					// Filebuffer Offset increment
					pstSysInfo^.stFileHandler.udiTmpFileBufferOffset := pstSysInfo^.stFileHandler.udiTmpFileBufferOffset + pstSysInfo^.udiTmpRecordLen;
					
					// clear temp. record buffer
					pstSysInfo^.bolTmpRecordFull := FALSE;
					
					// Record Buffer ist frei -> Offset zu Null setzen
					pstSysInfo^.udiTmpRecordLen := 0;
				END_IF
			ELSE // file buffer + temp record buffer exceeds maximum
				pstSysInfo^.stFileHandler.udiWriteTimer := 0; // reset timer
				pstSysInfo^.stFileHandler.usiCmd := FileLc.cCMD_FLUSHBUF; // write file buffer to file
			END_IF
		END_IF
		
		// return if buffer still full
		IF (pstSysInfo^.bolTmpRecordFull) THEN
			RETURN;
		END_IF
			

		// reset flag
		bolWriteRecord := FALSE;
		
		// Read out from base log -> stData
		uinReadStatus := stFileLogClientLibInfo.p_fbBasLog^.M_Read(In_pHandle:=pstSysInfo^.pBaseLogHandle,In_pData:=ADR(stData)); 
		IF (uinReadStatus<>0) THEN // exit for if nothing to read
			RETURN;
		END_IF
	
		// base logging
		IF(pstSysInfo^.uinLogTyp=FileLc.cLOGTYP_BL) THEN
			//reference item list
			pstItemCfgList := pstSysInfo^.stItemInfo.p_bytItemCfgList;
			
			// on BL only use first line
			pstItemDataList := pstSysInfo^.stItemInfo.a_p_bytItemDataList[0];
			
			// must be worked on the PvId ?
			 FOR jj := 0 TO (pstSysInfo^.stItemInfo.uinActNbrOfItems-1) BY 1 DO
				 CASE (pstItemCfgList[jj].dinPvId) OF
					FileLc.cPVTYPE_BL_LOGTYP:
						M_WriteActItemIdx(In_pstItemDataList :=pstItemDataList,In_dinDataTyp:= FileLc.cVAR_TYPE_UDINT, In_pValue:=ADR(stData.udiLogType), In_udiRecIdx:=0, In_uinActItemIdx:=jj);
					FileLc.cPVTYPE_BL_CTRL_ID:
						M_WriteActItemIdx(In_pstItemDataList :=pstItemDataList,In_dinDataTyp:= FileLc.cVAR_TYPE_INT, In_pValue:=ADR(stData.intCtrlID), In_udiRecIdx:=0, In_uinActItemIdx:=jj);
					FileLc.cPVTYPE_BL_STRING1:
						M_WriteActItemIdx(In_pstItemDataList :=pstItemDataList,In_dinDataTyp:= FileLc.cVAR_TYPE_STRING, In_pValue:=ADR(stData.strText1), In_udiRecIdx:=0, In_uinActItemIdx:=jj);
					FileLc.cPVTYPE_BL_STRING2:
						M_WriteActItemIdx(In_pstItemDataList :=pstItemDataList,In_dinDataTyp:= FileLc.cVAR_TYPE_STRING, In_pValue:=ADR(stData.strText2), In_udiRecIdx:=0, In_uinActItemIdx:=jj);
					FileLc.cPVTYPE_BL_PAR1:
						M_WriteActItemIdx(In_pstItemDataList :=pstItemDataList,In_dinDataTyp:= FileLc.cVAR_TYPE_DINT, In_pValue:=ADR(stData.dinPar1), In_udiRecIdx:=0, In_uinActItemIdx:=jj);
					FileLc.cPVTYPE_BL_PAR2:
						M_WriteActItemIdx(In_pstItemDataList :=pstItemDataList,In_dinDataTyp:= FileLc.cVAR_TYPE_DINT, In_pValue:=ADR(stData.dinPar2), In_udiRecIdx:=0, In_uinActItemIdx:=jj);
					FileLc.cPVTYPE_BL_PAR3:
						M_WriteActItemIdx(In_pstItemDataList :=pstItemDataList,In_dinDataTyp:= FileLc.cVAR_TYPE_DINT, In_pValue:=ADR(stData.dinPar3), In_udiRecIdx:=0, In_uinActItemIdx:=jj);
					FileLc.cPVTYPE_BL_PAR4:
						M_WriteActItemIdx(In_pstItemDataList :=pstItemDataList,In_dinDataTyp:= FileLc.cVAR_TYPE_DINT, In_pValue:=ADR(stData.dinPar4), In_udiRecIdx:=0, In_uinActItemIdx:=jj);
							
				END_CASE
			 END_FOR
			 // general inf o add to Record list
			pstSysInfo^.stItemInfo.stItemRecordData[0].dtActDateTime := stData.dtDateTimeEntry;
			pstSysInfo^.stItemInfo.stItemRecordData[0].uinActMilli := stData.uinMs;
			
			// for BaseLog write always record 0
			M_WriteRecord(In_pstSysInfo:=pstSysInfo,In_uinItemListIdx := 0);
			
			// end of IF(pstSysInfo^.uinLogTyp=FileLc.cLOGTYP_BL) THEN
		ELSE
			(* -----------------------------------*/
		  /* Data- und PV - Logging             */
		  /* -----------------------------------*)
	
		  (* ----------------------*/
		  /* Check commandes     */
		  /* ----------------------
		  /* "cmd" in typ field *)
		  IF (stData.dinPar3 = BasLog.cVAR_TYPE_CMD_NEW_REC) THEN
	
				(* search free record - list *)
				FOR jj := 0 TO Queue.cMAX_NR_OF_TASKS BY 1 DO
				  IF ((pstSysInfo^.stItemInfo.stItemRecordData[jj].udiRecIdx = 0) OR (DINT_TO_UDINT(stData.dinPar4) = pstSysInfo^.stItemInfo.stItemRecordData[jj].udiRecIdx)) THEN
						pstSysInfo^.stItemInfo.stItemRecordData[jj].udiRecIdx := DINT_TO_UDINT(stData.dinPar4);
						pstSysInfo^.stItemInfo.stItemRecordData[jj].dtActDateTime := stData.dtDateTimeEntry;
						pstSysInfo^.stItemInfo.stItemRecordData[jj].uinActMilli := stData.uinMs;
						EXIT;
				  END_IF
			   END_FOR
		  
		  ELSIF (stData.dinPar3 = BasLog.cVAR_TYPE_CMD_END_REC) THEN
			bolWriteRecord := TRUE;
		  END_IF			
	
	
		  (* --------------------------------------------------------------*/
		  /* entry reached BaseLog message in record list */
		  /* --------------------------------------------------------------*)
		  M_PutPvIdInList(In_pstSysInfo := pstSysInfo, In_pstData := ADR(stData));
	
		  (* -----------------------------------------------------*/
		  /* write the complete record to the temporar buffer */
		  /* -----------------------------------------------------*)
		  IF (bolWriteRecord)  THEN
			FOR jj := 0 TO Queue.cMAX_NR_OF_TASKS BY 1 DO
			  (* Is the reached record index allready entried in referencelist *)
			  IF (pstSysInfo^.stItemInfo.stItemRecordData[jj].udiRecIdx = DINT_TO_UDINT(stData.dinPar4)) THEN
				M_WriteRecord(In_pstSysInfo:=pstSysInfo,In_uinItemListIdx := jj);
				EXIT;
			  END_IF
			END_FOR
		  END_IF
    END_IF // else
  END_FOR // FOR ii := 0 TO ((pstSysInfo^.stItemInfo.uinActNbrOfItems-1) * 20) BY 1 DO
END_IF 	//IF (pstSysInfo^.stItemInfo.uinActNbrOfItems>0) THEN
END_METHOD

METHOD PUBLIC M_Init : BOOL
VAR_INPUT
	In_strCfgFileName: STRING(FileLc.cFILENAME_LENGTH); // name of the config/template file
	In_strPath: STRING(FileLc.cPATH_LENGTH);  // path of the config/template file
	In_p_fbBasLog: POINTER TO FB_BasLog; // only one central FB_BasLog instance allowed per PLC!!!
	In_bolExecute : BOOL;
	In_p_uinFLcIdx : POINTER TO UINT; // actual file client id
END_VAR
VAR_OUTPUT
	Out_pHandle: POINTER TO T_FileLc_SysInfo; // handle for cyclic call	
	Out_udiStatus: UDINT; 	// 0 => successful done, <>0 => error
	Out_bolDone: BOOL;		// Done
END_VAR

VAR
	strClientName : STRING(255);
	uinFLcIdxForArr : UINT;
	udiStatus : UDINT;
	udiMask : UDINT;
	uinInitStatus : UINT;
	pQueueInfoHandle : POINTER TO POINTER TO T_Queue_Info;
	fbGETCURTASKINDEX: Tc2_System.GETCURTASKINDEX;
	udiTaskCnt : UDINT;
END_VAR
// only one client init at the same on PLC possibel!!!
IF (In_p_uinFLcIdx<>Tc3_MemMan.NULL) THEN // valid actual id reference
	IF (In_bolExecute=TRUE) THEN
		// wait until release init rom other clients...
		IF  ((stFileLogClientLibInfo.uinActClientInitActive=0) OR (stFileLogClientLibInfo.uinActClientInitActive=In_p_uinFLcIdx^)) THEN
			IF (stFileLogClientLibInfo.uinActClientInitActive=0) THEN
				stFileLogClientLibInfo.uinActClientInitActive := stFileLogClientLibInfo.uinActNbrOfFileClients + 1; // lock init of other clients!!!
				In_p_uinFLcIdx^ := stFileLogClientLibInfo.uinActClientInitActive;
				
				Out_bolDone := 0;
				Out_udiStatus := 0;
				Out_pHandle := 0;
				//reset statemachine
				(* check input parameter *)
				IF (stFileLogClientLibInfo.uinActNbrOfFileClients >= FileLc.cMAX_NBR_OF_FILECLIENTS) THEN
					Out_udiStatus := FileLc.cERR_NBR_OF_FC_EXEEDED;
					RETURN;
				END_IF
				
				IF (In_strCfgFileName='') THEN
					Out_udiStatus := FileLc.cERR_FILENAME_MISSING;
					RETURN;
				END_IF
				
				IF (In_strPath='') THEN
					Out_udiStatus := FileLc.cERR_PATH_MISSING;
					RETURN;
				END_IF
				
				IF (In_p_fbBasLog=TC3_MEMMAN.NULL) THEN
					Out_udiStatus := FileLc.cERR_NO_BASELOG;
					RETURN;
				END_IF
		
				stFileLogClientLibInfo.p_fbBasLog := In_p_fbBasLog;
				
				// actual client init
				stFileLogClientLibInfo.stSysInfo[stFileLogClientLibInfo.uinActNbrOfFileClients].stStatemachine.uinState := 1;
				stFileLogClientLibInfo.stSysInfo[stFileLogClientLibInfo.uinActNbrOfFileClients].stStatemachine.uinState_old := 0;
				stFileLogClientLibInfo.stSysInfo[stFileLogClientLibInfo.uinActNbrOfFileClients].fbFileLc_WorkOnFile(In_bolExecute:=FALSE); // reset statemachine on next positive edge!
				
				// increment client number
				stFileLogClientLibInfo.uinActNbrOfFileClients := stFileLogClientLibInfo.uinActNbrOfFileClients + 1;
				
				
			END_IF
		
			// valid client idx
			IF (In_p_uinFLcIdx^>0) THEN
				uinFLcIdxForArr := In_p_uinFLcIdx^-1; // access idx for arrays!
			
				CASE stFileLogClientLibInfo.stSysInfo[uinFLcIdxForArr].stStatemachine.uinState OF
					1:
						// check template/config file */
						stFileLogClientLibInfo.stSysInfo[uinFLcIdxForArr].fbFileLc_WorkOnFile(In_bolExecute:=TRUE,In_strPath:=In_strPath,In_strCfgFileName:=In_strCfgFileName,In_pstSysInfo := ADR(stFileLogClientLibInfo.stSysInfo[uinFLcIdxForArr]));
						IF (stFileLogClientLibInfo.stSysInfo[uinFLcIdxForArr].fbFileLc_WorkOnFile.Out_udiStatus<>0) OR (stFileLogClientLibInfo.stSysInfo[uinFLcIdxForArr].fbFileLc_WorkOnFile.Out_bolDone=1) THEN
							stFileLogClientLibInfo.stSysInfo[uinFLcIdxForArr].stStatemachine.uinState := 2;
						END_IF
						
					2:
						IF (stFileLogClientLibInfo.stSysInfo[uinFLcIdxForArr].fbFileLc_WorkOnFile.Out_udiStatus<>0) THEN // error in template/config file
							stFileLogClientLibInfo.uinActNbrOfFileClients := stFileLogClientLibInfo.uinActNbrOfFileClients - 1;
							Out_udiStatus := stFileLogClientLibInfo.stSysInfo[uinFLcIdxForArr].fbFileLc_WorkOnFile.Out_udiStatus;
							RETURN;
						END_IF
						  
						// register as client on base log system
						strClientName := BasLog.cCLIENT_NAME_PF;
						strClientName := Tc2_Standard.CONCAT(strClientName,'.fileclient');
						strClientName := Tc2_Standard.CONCAT(strClientName,UINT_TO_STRING(uinFLcIdxForArr));
						
						//LOG TYPE Maske --> PVLog Event und Cyclic 
						CASE (stFileLogClientLibInfo.stSysInfo[uinFLcIdxForArr].uinLogTyp) OF
							FileLc.cLOGTYP_DATA:
								udiMask := BasLog.cLOGTYPE_DATA;
							FileLc.cLOGTYP_PV:
								udiMask := (BasLog.cLOGTYPE_PV_EVENT OR BasLog.cLOGTYPE_PV_CYCLIC);
							FileLc.cLOGTYP_BL, FileLc.cLOGTYP_OPEN:
								udiMask := stFileLogClientLibInfo.stSysInfo[uinFLcIdxForArr].udiMask;
						END_CASE
						
						stFileLogClientLibInfo.fbTimeStamp.In_strNetId := stFileLogClientLibInfo.stSysInfo[uinFLcIdxForArr].stConfig.strLogNetId; // use system time of log target system
						stFileLogClientLibInfo.fbTimeStamp.In_t_CycleTimeRefreshTimeZone := T#0S; // cyclic check time zone settings - not needed using LocalTime_FileTime_BaseWin for log system and local time
						stFileLogClientLibInfo.p_fbBasLog^.M_ClientInit(In_strClientName:=strClientName,In_udiMask := udiMask, In_uinNrOfElement:= UDINT_TO_UINT(stFileLogClientLibInfo.stSysInfo[uinFLcIdxForArr].stConfig.udiQueueLen),In_p_fbTimeStamp:=ADR(stFileLogClientLibInfo.fbTimeStamp),In_bolUseLocalTimeStamp:=stFileLogClientLibInfo.stSysInfo[uinFLcIdxForArr].stConfig.bolUseLocalTimeStamp,Out_pHandle=>pQueueInfoHandle,Out_uinStatus=>udiStatus);
						
						IF (udiStatus<>0) THEN // check if init base log ok
							stFileLogClientLibInfo.uinActNbrOfFileClients := stFileLogClientLibInfo.uinActNbrOfFileClients - 1;
							Out_udiStatus := udiStatus;
							RETURN;
						END_IF
				
						//---------------------------------------------------------------------------------------------------------------
						// set SysInfo parameter
						stFileLogClientLibInfo.stSysInfo[uinFLcIdxForArr].pBaseLogHandle := pQueueInfoHandle;
						//DeviceName auf SysInfo Struktur ablegen
						stFileLogClientLibInfo.stSysInfo[uinFLcIdxForArr].strPathName := In_strPath;
						
						// get cycle time
						// number of tasksudiTaskCnt := TwinCAT_SystemInfoVarList._AppInfo.TaskCnt;
						fbGETCURTASKINDEX();
						udiTaskCnt := fbGETCURTASKINDEX.index;
						stFileLogClientLibInfo.stSysInfo[uinFLcIdxForArr].udiCylceTimeMs := TwinCAT_SystemInfoVarList._TaskInfo[UDINT_TO_DINT(udiTaskCnt)].CycleTime/10000; //[ms] X[100ns]/10000 -> [ms]
			
						// init filehandler
						//automatic read out infos about FUB
						udiStatus := stFileLogClientLibInfo.stSysInfo[uinFLcIdxForArr].stFileHandler.FB_FileLc_FileHdl.M_Init(In_pstSysInfo:=ADR(stFileLogClientLibInfo.stSysInfo[uinFLcIdxForArr]));
						IF (udiStatus<>0) THEN // check if init base log ok
							stFileLogClientLibInfo.uinActNbrOfFileClients := stFileLogClientLibInfo.uinActNbrOfFileClients - 1;
							Out_udiStatus := udiStatus;
							RETURN;
						END_IF
						
						// finished
						stFileLogClientLibInfo.stSysInfo[uinFLcIdxForArr].stStatemachine.uinState := 3;
					3:
						// wait for time stamp init ok (synchronize windows time, get time zone information!)
						stFileLogClientLibInfo.fbTimeStamp();
						IF (stFileLogClientLibInfo.fbTimeStamp.Out_bolInitOk) THEN
							stFileLogClientLibInfo.stSysInfo[uinFLcIdxForArr].stStatemachine.uinState := 4;
						END_IF
					4: 
						stFileLogClientLibInfo.stSysInfo[uinFLcIdxForArr].stStatemachine.usiInitDone := 1;
						Out_bolDone := TRUE; // init done
						stFileLogClientLibInfo.uinActClientInitActive := 0; // release init of other clients!!!
						// return adresse on actual SysInfo struct
						Out_pHandle := ADR(stFileLogClientLibInfo.stSysInfo[uinFLcIdxForArr]);
				END_CASE
			END_IF
		END_IF
	ELSE
		IF (stFileLogClientLibInfo.uinActClientInitActive=In_p_uinFLcIdx^) THEN // reset own flag
			stFileLogClientLibInfo.uinActClientInitActive := 0; // release init of other clients!!!
		END_IF
	END_IF
ELSE
	Out_pHandle := 0;
	Out_udiStatus := FileLc.cERR_NO_FLCIDX;
	RETURN;
END_IF
END_METHOD

METHOD PROTECTED M_PutPvIdInList : UINT
VAR_INPUT
	In_pstSysInfo: POINTER TO T_FileLc_SysInfo;
	In_pstData : POINTER TO T_Bl_BaseStruc;
END_VAR
VAR
	pstItemDataList : POINTER TO T_FileLc_ItemData;
  	pstItemCfgList: POINTER TO T_FileLc_ItemCfg;
	pstItemCfgListItem: T_FileLc_ItemCfg;
	bolItemFound : BOOL;
	uinActItemIdx : UINT;
	ii: UINT;
END_VAR
// Methode check received base log message and fill up the data to the item list
pstItemCfgList := In_pstSysInfo^.stItemInfo.p_bytItemCfgList;

bolItemFound := FALSE;

// has the id to be overworked?
FOR ii := 0 TO (In_pstSysInfo^.stItemInfo.uinActNbrOfItems-1) BY 1 DO
	pstItemCfgListItem := pstItemCfgList[ii];
	IF (pstItemCfgList[ii].dinPvId=In_pstData^.dinPar1) THEN
	 	bolItemFound := TRUE;
		uinActItemIdx := ii;
		EXIT;
	END_IF
END_FOR

// this PvId is not in list
IF (bolItemFound=FALSE) THEN
	M_PutPvIdInList := 0;
	RETURN;
END_IF

(* ---------------------------------*/
/* check reference list      */
/* and write data to the list */
/* ---------------------------------*)
FOR ii := 0 TO Queue.cMAX_NR_OF_TASKS BY 1 DO

	(* Is the received record in reference list?*)
	IF (In_pstSysInfo^.stItemInfo.stItemRecordData[ii].udiRecIdx = DINT_TO_UDINT(In_pstData^.dinPar4)) THEN
			
	  // reference to item list
	  pstItemDataList := In_pstSysInfo^.stItemInfo.a_p_bytItemDataList[ii];
	
	  (* write data to item list *)
	  IF (In_pstData^.dinPar3 = FileLc.cVAR_TYPE_STRING) THEN// data definition
		M_WriteActItemIdx(In_pstItemDataList :=pstItemDataList,In_dinDataTyp:= FileLc.cVAR_TYPE_STRING, In_pValue:=ADR(In_pstData^.strText2), In_udiRecIdx:=DINT_TO_UDINT(In_pstData^.dinPar4), In_uinActItemIdx:=uinActItemIdx);
	  ELSE
		M_WriteActItemIdx(In_pstItemDataList:=pstItemDataList, In_dinDataTyp := In_pstData^.dinPar3, In_pValue := ADR(In_pstData^.dinPar2),In_udiRecIdx := DINT_TO_UDINT(In_pstData^.dinPar4), In_uinActItemIdx := uinActItemIdx);
	  END_IF
	  EXIT;
	END_IF
END_FOR		

M_PutPvIdInList := 0;
RETURN;
END_METHOD

METHOD PROTECTED M_ReleaseBuffer : UINT

VAR_INPUT
	In_pReleaseBuffer : POINTER TO BYTE;
END_VAR
//delocate  allocated buffer with __NEW
__DELETE(In_pReleaseBuffer);
RETURN; // delete buffer with dynamic size...
END_METHOD

METHOD PROTECTED M_WriteActItemIdx : UINT
VAR_INPUT
	In_pstItemDataList : POINTER TO T_FileLc_ItemData;
	In_dinDataTyp: DINT;
	In_pValue: POINTER TO BYTE;
	In_udiRecIdx : UDINT;
	In_uinActItemIdx : UINT;
END_VAR

VAR
	strTmp : T_MaxString;
	pString : POINTER TO STRING(255);
	pBool : POINTER TO BOOL;
	pSint : POINTER TO SINT;
	pInt : POINTER TO INT;
	pDint : POINTER TO DINT;
	pUsint : POINTER TO USINT;
	pUint : POINTER TO UINT;
	pUdint : POINTER TO UDINT;
	pReal : POINTER TO REAL;
	pLreal : POINTER TO LREAL;
	stItemDataListItem : T_FileLc_ItemData;
END_VAR
// write value in ItemList based on datatyp
IF (In_pValue<>TC3_MEMMAN.NULL) THEN
	 CASE In_dinDataTyp OF
		FileLc.cVAR_TYPE_SINT:
			pSint := In_pValue;
			strTmp := SINT_TO_STRING(pSint^);	
		FileLc.cVAR_TYPE_INT:
			pInt := In_pValue;
			strTmp := INT_TO_STRING(pInt^);
		FileLc.cVAR_TYPE_DINT:
			pDint := In_pValue;
			strTmp := DINT_TO_STRING(pDint^);
		FileLc.cVAR_TYPE_BOOL:
			pBool := In_pValue;
			strTmp := BOOL_TO_STRING(pBool^);	
		FileLc.cVAR_TYPE_USINT:
			pUsint := In_pValue;
			strTmp := USINT_TO_STRING(pUsint^);
		FileLc.cVAR_TYPE_UINT:
			pUint := In_pValue;
			strTmp := UINT_TO_STRING(pUint^);
		FileLc.cVAR_TYPE_UDINT:
			pUdint := In_pValue;
			strTmp := UDINT_TO_STRING(pUdint^);
		FileLc.cVAR_TYPE_REAL:
			pReal := In_pValue;
			strTmp := REAL_TO_STRING(pReal^);
		FileLc.cVAR_TYPE_LREAL:
			pLreal := In_pValue;
			strTmp := LREAL_TO_STRING(pLreal^);
		FileLc.cVAR_TYPE_STRING:
			pString := In_pValue;
			strTmp := pString^;
		ELSE
			strTmp := 'unknown type';
	END_CASE
	
	IF (INT_TO_UINT(LEN(strTmp)) >=  FileLc.cMAX_ITEM_CHAR) THEN
		In_pstItemDataList[In_uinActItemIdx].strValue:= 'value too long';
	ELSE
		MEMSET(destAddr := ADR(In_pstItemDataList[In_uinActItemIdx].strValue),0,SIZEOF(In_pstItemDataList[In_uinActItemIdx].strValue)); // string ends wit 0!
		MEMCPY(destAddr := ADR(In_pstItemDataList[In_uinActItemIdx].strValue),srcAddr:=ADR(strTmp),SIZEOF(strTmp));
	END_IF
END_IF
// entry record index
In_pstItemDataList[In_uinActItemIdx].udiRecIdx := In_udiRecIdx;
stItemDataListItem := In_pstItemDataList[In_uinActItemIdx]; // for Debugging
END_METHOD

METHOD PROTECTED M_WriteRecord : UINT
VAR_INPUT
	In_pstSysInfo: POINTER TO T_FileLc_SysInfo;
	In_uinItemListIdx : UINT;
END_VAR
VAR
 	pstItemDataList : POINTER TO T_FileLc_ItemData;
  	pstItemCfgList: POINTER TO T_FileLc_ItemCfg;
	pstItemCfgListItem: T_FileLc_ItemCfg;
	pstItemDataListItem : T_FileLc_ItemData;
	pstRecordData : POINTER TO T_FileLc_RecordData;
	ii : UINT;
	bolRecordValid : BOOL;
	udiOffset : UDINT;
	udiTmpLen : UDINT;
	strTemp : STRING(30);
	SystemTimeStruct  :TIMESTRUCT;
END_VAR
pstItemDataList := In_pstSysInfo^.stItemInfo.a_p_bytItemDataList[In_uinItemListIdx];
pstItemCfgList := In_pstSysInfo^.stItemInfo.p_bytItemCfgList;
pstRecordData := ADR(In_pstSysInfo^.stItemInfo.stItemRecordData[In_uinItemListIdx]);

// copy PRE - Text
udiOffset := 0;
udiTmpLen := INT_TO_UDINT(LEN(In_pstSysInfo^.stItemInfo.strPreItemText));
MEMCPY(destAddr := (In_pstSysInfo^.p_bytTmpRecordText+udiOffset),srcAddr :=ADR(In_pstSysInfo^.stItemInfo.strPreItemText) , n := udiTmpLen);
udiOffset := udiOffset + udiTmpLen;

// check filled data
bolRecordValid := FALSE;
//at least one item has to be added before
FOR ii := 0 TO (In_pstSysInfo^.stItemInfo.uinActNbrOfItems-1) BY 1 DO
	pstItemCfgListItem := pstItemCfgList[ii];
	pstItemDataListItem := pstItemDataList[ii];
	IF ((pstItemCfgListItem.dinPvId>=0) AND (pstItemDataListItem.udiRecIdx=pstRecordData^.udiRecIdx)) THEN
	 	bolRecordValid := TRUE;
		 EXIT;
	END_IF
END_FOR

// record has no valid data
IF ((bolRecordValid=FALSE) AND (In_pstSysInfo^.uinLogTyp<>FileLc.cLOGTYP_BL)) THEN
	// clear record data
	pstRecordData^.udiRecIdx :=0;
	pstRecordData^.dtActDateTime := REAL_TO_DT(0.0);
	pstRecordData^.uinActMilli :=0;
	
	// reset record buffer
	In_pstSysInfo^.udiTmpRecordLen := 0;
	In_pstSysInfo^.bolTmpRecordFull := FALSE;
	RETURN;
END_IF

// collect data
FOR ii := 0 TO (In_pstSysInfo^.stItemInfo.uinActNbrOfItems-1) BY 1 DO
	//for debugging
	pstItemCfgListItem := pstItemCfgList[ii];
	pstItemDataListItem := pstItemDataList[ii];
	
	IF (pstItemCfgListItem.dinPvId<0) THEN
	 	CASE (pstItemCfgListItem.dinPvId) OF
			FileLc.cPVTYPE_UNIX_DATE_TIME_STR:
				// time and date as string
				pstItemDataListItem.strValue := DT_TO_STRING(pstRecordData^.dtActDateTime);
			
			FileLc.cPVTYPE_UNIX_DATE_TIME:
				// time and date as  s since 1.1.1970 11:00
				pstItemDataListItem.strValue := DWORD_TO_STRING(DT_TO_DWORD(pstRecordData^.dtActDateTime));
			
			FileLc.cPVTYPE_EXCEL_DATE_TIME:
				// time and date as REAL
				pstItemDataListItem.strValue := LREAL_TO_STRING(DT_TO_LREAL(pstRecordData^.dtActDateTime));
				(*needed ?? if (pdstRecordData->dtActDateTime > 0) {
						tmpDouble = (double)(pdstRecordData->dtActDateTime / 86400.0) + 25569.0;
						tmpUdint = (double)tmpDouble;  /*Ganzzahl bilden/
						tmpDouble = (tmpDouble - tmpUdint); /*Nachkommastellen/
						itoa(tmpUdint, (unsigned long)&pdstItemDataList[i].strValue);
						strcat((void)&pdstItemDataList[i].strValue, ".");

						// Nachkommaanteil mit 10 hoch n multipizieren
						tmpUdint = tmpDouble * tmpPrecision;
	
						// Integer to ACSI Wandlung mit Vornullen!
						tmpPrecision = tmpPrecision / 10;
						n=0;
						while (tmpPrecision > 1) {
							tmpString[n] = (tmpUdint / tmpPrecision) + 0x30;  // Character Wandlung
							tmpUdint = tmpUdint % tmpPrecision;
							tmpPrecision = tmpPrecision / 10;
							n++;
						}
						tmpString[n]=0;
						strcat((void)&pdstItemDataList[i].strValue, (void)&tmpString);
						ulSize = strlen(pdstItemDataList[i].strValue);
					}*)
			FileLc.cPVTYPE_DATE_SLASH_TIME_COLON: 
				//english date format 2014/09/23 07:10:24
				SystemTimeStruct := DT_TO_SYSTEMTIME(pstRecordData^.dtActDateTime);
				pstItemDataListItem.strValue := DWORD_TO_STRING(SystemTimeStruct.wYear);
				pstItemDataListItem.strValue := CONCAT(STR1:=pstItemDataListItem.strValue,STR2:='/');
				IF (SystemTimeStruct.wMonth<10) THEN
					pstItemDataListItem.strValue := CONCAT(pstItemDataListItem.strValue , '0');
				END_IF
				pstItemDataListItem.strValue := CONCAT(STR1:=pstItemDataListItem.strValue,STR2:=DWORD_TO_STRING(SystemTimeStruct.wMonth));
				pstItemDataListItem.strValue := CONCAT(STR1:=pstItemDataListItem.strValue,STR2:='/');
				IF (SystemTimeStruct.wDay<10) THEN
					pstItemDataListItem.strValue := CONCAT(pstItemDataListItem.strValue , '0');
				END_IF
				pstItemDataListItem.strValue := CONCAT(STR1:=pstItemDataListItem.strValue,STR2:=DWORD_TO_STRING(SystemTimeStruct.wDay));
				pstItemDataListItem.strValue := CONCAT(STR1:=pstItemDataListItem.strValue,STR2:=' ');
				IF (SystemTimeStruct.wHour<10) THEN
					pstItemDataListItem.strValue := CONCAT(pstItemDataListItem.strValue , '0');
				END_IF
				pstItemDataListItem.strValue := CONCAT(STR1:=pstItemDataListItem.strValue,STR2:=DWORD_TO_STRING(SystemTimeStruct.wHour));
				pstItemDataListItem.strValue := CONCAT(STR1:=pstItemDataListItem.strValue,STR2:=':');
				IF (SystemTimeStruct.wMinute<10) THEN
					pstItemDataListItem.strValue := CONCAT(pstItemDataListItem.strValue , '0');
				END_IF
				pstItemDataListItem.strValue := CONCAT(STR1:=pstItemDataListItem.strValue,STR2:=DWORD_TO_STRING(SystemTimeStruct.wMinute));
				pstItemDataListItem.strValue := CONCAT(STR1:=pstItemDataListItem.strValue,STR2:=':');
				IF (SystemTimeStruct.wSecond<10) THEN
					pstItemDataListItem.strValue := CONCAT(pstItemDataListItem.strValue , '0');
				END_IF
				pstItemDataListItem.strValue := CONCAT(STR1:=pstItemDataListItem.strValue,STR2:=DWORD_TO_STRING(SystemTimeStruct.wSecond));
			FileLc.cPVTYPE_TIME_MILLI:
				IF (pstRecordData^.uinActMilli<100) THEN
					IF (pstRecordData^.uinActMilli<10) THEN
						pstItemDataListItem.strValue := '00';
					ELSE
						pstItemDataListItem.strValue := '0';
					END_IF
				ELSE
					pstItemDataListItem.strValue := '';
				END_IF
				pstItemDataListItem.strValue := CONCAT(STR1:=pstItemDataListItem.strValue,STR2:=UINT_TO_STRING(pstRecordData^.uinActMilli));
		END_CASE
	END_IF
	
	
	(* ----------------------------------*/ 
	/* Write data to temp buffer */
	/* ----------------------------------*/ 
	/* PV value *)		
	IF ((pstItemDataListItem.udiRecIdx = pstRecordData^.udiRecIdx) OR (pstItemCfgListItem.dinPvId < 0)) THEN
		udiTmpLen := INT_TO_UDINT(LEN(pstItemDataListItem.strValue));
		MEMCPY(destAddr := (In_pstSysInfo^.p_bytTmpRecordText+udiOffset),srcAddr :=ADR(pstItemDataListItem.strValue) , n := udiTmpLen);
	ELSE 
		strTemp := 'no val.';
		udiTmpLen := INT_TO_UDINT(LEN(strTemp)); 
		MEMCPY(destAddr := (In_pstSysInfo^.p_bytTmpRecordText+udiOffset),srcAddr :=ADR(strTemp) , n := udiTmpLen);	
	END_IF
	udiOffset := udiOffset + udiTmpLen;
	
	IF (ii>0) AND (ii=In_pstSysInfo^.stItemInfo.uinActNbrOfItems-1) AND (udiTmpLen=0) THEN // last text empty...
		// remove last post text...
		udiTmpLen := INT_TO_UDINT(LEN(pstItemCfgList[ii-1].strPostText));
		IF (udiOffset>udiTmpLen) THEN
			MEMSET(destAddr := (In_pstSysInfo^.p_bytTmpRecordText+udiOffset-udiTmpLen),fillByte :=0 , n := udiTmpLen);
			udiOffset := udiOffset - udiTmpLen;
		END_IF
	END_IF
	
	(* Post Text *)	
	udiTmpLen := INT_TO_UDINT(LEN(pstItemCfgListItem.strPostText));
	MEMCPY(destAddr := (In_pstSysInfo^.p_bytTmpRecordText+udiOffset),srcAddr :=ADR(pstItemCfgListItem.strPostText) , n := udiTmpLen);
	udiOffset := udiOffset + udiTmpLen;

END_FOR(*for (i = 0; i < pdstSysInfo->dstItemInfo.uinActNbrOfItems; i++) *)


(* carriage return on end of record *)
udiTmpLen := SIZEOF(FileLc.cEOL);
MEMCPY(destAddr := (In_pstSysInfo^.p_bytTmpRecordText+udiOffset),srcAddr :=ADR(FileLc.cEOL) , n := udiTmpLen);
udiOffset := udiOffset + udiTmpLen;

// clear record data
pstRecordData^.udiRecIdx :=0;
pstRecordData^.dtActDateTime :=REAL_TO_DT(0.0);
pstRecordData^.uinActMilli :=0;

// mark record buffer as full
In_pstSysInfo^.udiTmpRecordLen := udiOffset;
In_pstSysInfo^.bolTmpRecordFull := TRUE;

(*--------------------------------*/
/* count file entries */
/*--------------------------------*)
In_pstSysInfo^.stFileHandler.udiRecordCnt := In_pstSysInfo^.stFileHandler.udiRecordCnt + 1;
END_METHOD

END_FUNCTION_BLOCK

// POUs/Utility/Logger/FileLc/FB_FileLc_FileHdl
FUNCTION_BLOCK FB_FileLc_FileHdl
VAR_INPUT
END_VAR
VAR_OUTPUT
END_VAR
VAR
	fbFileHdl : FB_FileHdl;
	bol_fpNewFileEvent : BOOL;
END_VAR

PROPERTY PUBLIC ActFileSize : UDINT
GET
ActFileSize := fbFileHdl.ActFileSize;
END_GET
END_PROPERTY

METHOD PUBLIC M_Cyclic : UDINT
VAR_INPUT
	In_pstSysInfo: POINTER TO T_FileLc_SysInfo;
END_VAR

VAR

END_VAR
VAR CONSTANT
	// specific steps definitions
	cStep_Wait4Job: UINT := 500;
	cStep_WriteFileBuf: UINT := 501;
	cStep_WriteFooter: UINT := 502;
	cStep_CreateNew: UINT := 503;
	cStep_WriteHeader: UINT := 504;
END_VAR
fbFileHdl();

CASE In_pstSysInfo^.stFileHandler.uinState OF
	0:	In_pstSysInfo^.stFileHandler.uinState := cStep_Wait4Job;
	
	// ready for new job
	cStep_Wait4Job:
		IF (In_pstSysInfo^.stFileHandler.uinState<>In_pstSysInfo^.stFileHandler.uinState_old) THEN
			In_pstSysInfo^.stFileHandler.strInfo := 'I: cStep_Wait4Job';
			
			In_pstSysInfo^.stFileHandler.uinState_old := In_pstSysInfo^.stFileHandler.uinState;
		END_IF
		
		// file handler ready for new commands
		IF (fbFileHdl.Out_bolBusy=FALSE) THEN
			// create new file after startup
			IF ((In_pstSysInfo^.stConfig.uinNewFileOnRestart=1) AND (In_pstSysInfo^.stFileHandler.usiInitDone=0)) THEN
				In_pstSysInfo^.stFileHandler.usiCmdNewFile := 1; 
			END_IF
			
			// mark for restart detection
			In_pstSysInfo^.stFileHandler.usiInitDone := 1;	

			// event from filehandler nwe file created!!!
			IF (fbFileHdl.Out_bolNewFileCreated) THEN
				IF (bol_fpNewFileEvent=FALSE) THEN // detect positive edge on signal!!
					bol_fpNewFileEvent := TRUE;
					In_pstSysInfo^.stFileHandler.uinState := cStep_WriteHeader;
				END_IF
			ELSE
				bol_fpNewFileEvent := FALSE;
			END_IF
			
			// finish file
			IF (In_pstSysInfo^.stFileHandler.usiCmdNewFile=1) THEN
				In_pstSysInfo^.stFileHandler.usiCmd := FileLc.cCMD_FLUSHBUF_NEWFILE;
				In_pstSysInfo^.stFileHandler.usiCmdNewFile :=0;
			END_IF
			
			// temp file buffer write to file
			IF ((In_pstSysInfo^.stFileHandler.usiCmd=FileLc.cCMD_FLUSHBUF_NEWFILE) OR (In_pstSysInfo^.stFileHandler.usiCmd=FileLc.cCMD_FLUSHBUF)) THEN
				In_pstSysInfo^.stFileHandler.uinState :=cStep_WriteFileBuf;
				
			END_IF
		END_IF
	
	// write file buffer to file
	cStep_WriteFileBuf:
		// entry action
		IF (In_pstSysInfo^.stFileHandler.uinState<>In_pstSysInfo^.stFileHandler.uinState_old) THEN
			In_pstSysInfo^.stFileHandler.strInfo := 'I: cStep_WriteFileBuf';
			
			fbFileHdl.M_Cmd_WriteBuffer(In_p_bytWriteBuff:=In_pstSysInfo^.stFileHandler.p_bytTmpFileBuffer,In_udiWriteLen:=In_pstSysInfo^.stFileHandler.udiTmpFileBufferOffset);
			fbFileHdl(); // first call -> set busy flag = TRUE
			
			In_pstSysInfo^.stFileHandler.uinState_old := In_pstSysInfo^.stFileHandler.uinState;
		END_IF
		
		fbFileHdl(); // first call -> set busy flag = TRUE
		
		// always action
		IF (fbFileHdl.Out_bolBusy=FALSE) THEN
			IF (fbFileHdl.Out_udiErrId<>0) THEN
				In_pstSysInfo^.stFileHandler.usiCmd := 0;
				In_pstSysInfo^.stFileHandler.uinState :=cStep_WriteFooter;
			ELSIF (In_pstSysInfo^.stFileHandler.usiCmd=FileLc.cCMD_FLUSHBUF) THEN
				// reset file buffer and add offset
				In_pstSysInfo^.stFileHandler.udiTmpFileBufferOffset := 0;
				In_pstSysInfo^.stFileHandler.usiCmd := 0;
				In_pstSysInfo^.stFileHandler.uinState :=cStep_Wait4Job;
			ELSIF (In_pstSysInfo^.stFileHandler.usiCmd=FileLc.cCMD_FLUSHBUF_NEWFILE) THEN
				// reset file buffer and add offset
				In_pstSysInfo^.stFileHandler.udiTmpFileBufferOffset := 0;
				In_pstSysInfo^.stFileHandler.uinState :=cStep_WriteFooter;
			END_IF
		END_IF
		
	// write footer to file
	cStep_WriteFooter:
		// entry action
		IF (In_pstSysInfo^.stFileHandler.uinState<>In_pstSysInfo^.stFileHandler.uinState_old) THEN
			In_pstSysInfo^.stFileHandler.strInfo := 'I: cStep_WriteFooter';
			
			fbFileHdl.M_Cmd_WriteBuffer(In_p_bytWriteBuff:=In_pstSysInfo^.p_bytFooterText,In_udiWriteLen:=In_pstSysInfo^.udiFooterTextLen);
			fbFileHdl(); // first call -> set busy flag = TRUE
			
			In_pstSysInfo^.stFileHandler.uinState_old := In_pstSysInfo^.stFileHandler.uinState;
		END_IF
		
		fbFileHdl(); // first call -> set busy flag = TRUE
		
		// always action
		IF (fbFileHdl.Out_bolBusy=FALSE) THEN
			IF (fbFileHdl.Out_udiErrId<>0) THEN
				In_pstSysInfo^.stFileHandler.uinState :=cStep_CreateNew;
			ELSE
				In_pstSysInfo^.stFileHandler.uinState :=cStep_CreateNew;
			END_IF
		END_IF
		
	// create new file
	cStep_CreateNew:
		// entry action
		IF (In_pstSysInfo^.stFileHandler.uinState<>In_pstSysInfo^.stFileHandler.uinState_old) THEN
			In_pstSysInfo^.stFileHandler.strInfo := 'I: cStep_CreateNew';
			
			fbFileHdl.M_Cmd_NewFile();
			fbFileHdl(); // first call -> set busy flag = TRUE
			
			In_pstSysInfo^.stFileHandler.uinState_old := In_pstSysInfo^.stFileHandler.uinState;
		END_IF
		
		fbFileHdl(); // first call -> set busy flag = TRUE
		
		// always action
		IF (fbFileHdl.Out_bolBusy=FALSE) THEN
			In_pstSysInfo^.stFileHandler.uinState := cStep_WriteHeader;
		END_IF
		
	// create new file
	cStep_WriteHeader:
		// entry action
		IF (In_pstSysInfo^.stFileHandler.uinState<>In_pstSysInfo^.stFileHandler.uinState_old) THEN
			In_pstSysInfo^.stFileHandler.strInfo := 'I: cStep_WriteHeader';
			
			fbFileHdl.M_Cmd_WriteBuffer(In_p_bytWriteBuff:=In_pstSysInfo^.p_bytHeaderText,In_udiWriteLen:=In_pstSysInfo^.udiHeaderTextLen);
			fbFileHdl(); // first call -> set busy flag = TRUE
			
			In_pstSysInfo^.stFileHandler.uinState_old := In_pstSysInfo^.stFileHandler.uinState;
		END_IF
		
		fbFileHdl(); // first call -> set busy flag = TRUE
		
		// always action
		IF (fbFileHdl.Out_bolBusy=FALSE) THEN
			In_pstSysInfo^.stFileHandler.usiCmd := 0;
			In_pstSysInfo^.stFileHandler.uinState := cStep_Wait4Job;
		END_IF
END_CASE

fbFileHdl();

M_Cyclic := fbFileHdl.Out_udiErrId; // error number feedback, reset with next job
END_METHOD

METHOD PUBLIC M_Init : UDINT
VAR_INPUT
	In_pstSysInfo: POINTER TO T_FileLc_SysInfo;
END_VAR
// max file size set higher than defined because of writing footer before create new file -> FileLc manages max file size!!!
fbFileHdl.M_Init(In_strNetId := In_pstSysInfo^.stConfig.strLogNetId ,IN_strPath:= In_pstSysInfo^.stConfig.strLogPath,IN_strFileName:=In_pstSysInfo^.stConfig.strLogFileNamePraeFix,IN_strFileExt:=In_pstSysInfo^.stConfig.strLogFileNameExt,IN_uinMaxNrOfFilesInFolder:=In_pstSysInfo^.stConfig.uinMaxNbrOfLogFiles,IN_lreMaxFileSize:=(UDINT_TO_REAL(In_pstSysInfo^.stConfig.udiMaxFileSize)*1.2),IN_timFileSupervisionPeriod:=UDINT_TO_TIME(In_pstSysInfo^.stConfig.udiTimeCheckMaxFileNr));
M_Init := fbFileHdl.Out_udiErrId;
END_METHOD

END_FUNCTION_BLOCK

// POUs/Utility/Logger/FileLc/FB_FileLc_WorkOnFile
FUNCTION_BLOCK FB_FileLc_WorkOnFile
VAR_INPUT
	In_strCfgFileName: STRING(FileLc.cFILENAME_LENGTH); // name of the config/template file (not implemented yet)
	In_strPath: STRING(FileLc.cPATH_LENGTH); 
	In_pstSysInfo : POINTER TO T_FileLc_SysInfo;
	In_bolExecute : BOOL;
END_VAR
VAR_OUTPUT
	Out_udiStatus: UDINT;			// Rückgabewert 0:ok
	Out_bolDone: BOOL;			// Done
END_VAR
VAR
	fbFileOpen : FB_FileOpen;
	fbFileRead : FB_FileRead;
	fbFileClose : FB_FileClose;
	fbFileSeek : FB_FileSeek;
	udiWaitFileOpenCycles : UDINT;
	udiWaitFileReadCycles : UDINT;
	uinFileSize: UINT := 1000; // nr of Bytes to read whole config file
	p_bytTemplateBegin : POINTER TO BYTE;
	p_bytTemplateEnd : POINTER TO BYTE;
	p_bytConfigBegin : POINTER TO BYTE;
	p_bytConfigEnd : POINTER TO BYTE;
	p_bytHeaderBegin : POINTER TO BYTE;
	p_bytHeaderEnd : POINTER TO BYTE;
	p_bytFooterBegin : POINTER TO BYTE;
	p_bytFooterEnd : POINTER TO BYTE;
	p_bytRecordBegin : POINTER TO BYTE;
	p_bytRecordEnd : POINTER TO BYTE;
	p_bytTmpDestAdr : POINTER TO BYTE;
	p_bytTmpSrcAdr : POINTER TO BYTE;
	p_bytRowBegin : POINTER TO BYTE;
	p_bytRowEnd : POINTER TO BYTE;
	p_bytItemBegin : POINTER TO BYTE;
	p_bytItemEnd : POINTER TO BYTE;
	p_bytLastPos : POINTER TO BYTE;
	p_bytConfigValBegin : POINTER TO BYTE;
	p_bytConfigValEnd : POINTER TO BYTE;
	uinTmpLen : UINT;
	uinItemCount : UINT;
	ii : USINT;
	p_stItemCfgList : POINTER TO T_FileLc_ItemCfg;
	udiTmpLen : UDINT;
	strTmp : T_MaxString;
	udiWaitFileCloseCycles : UDINT := 0;
	bolBufferNotOk : BOOL;
	udiFileConfigLen : UDINT;
	pstrTmp : POINTER TO T_MaxString;
	strTmpTest:T_MaxString;
	stStatemachine : T_FileLc_Statemachine;
	strInfo :T_MaxString;
	bolExecute_old : BOOL;
	bolTmp : BOOL;
	pDelReadPointer : POINTER TO BYTE;
END_VAR

IF (In_bolExecute=TRUE) THEN
	IF (bolExecute_old=FALSE) THEN
		//reset statemachine
		stStatemachine.uinState :=0;
		stStatemachine.uinState_old := 255;
		Out_bolDone := 0;
		Out_udiStatus := 0;
	END_IF
	;
	
	CASE stStatemachine.uinState OF
		0: 
			IF (In_strCfgFileName<>'') THEN
				Out_bolDone := FALSE;
				strInfo := '';
				Out_udiStatus := 0;
				pstrTmp := ADR(strTmpTest);
				stStatemachine.uinState := stStatemachine.uinState  + 1;
			END_IF
		1: 
			// Entry action
			IF (stStatemachine.uinState_old <> stStatemachine.uinState) THEN
				//---------------------------------------------------------
				// File parser and check settings/configs
				//---------------------------------------------------------
				
				//*********************************************************
				// file open
				fbFileOpen.sNetId := ''; // only local access
				fbFileOpen.sPathName := CONCAT(STR1:=In_strPath,STR2:=In_strCfgFileName);
				fbFileOpen.nMode := Tc2_System.FOPEN_MODEREAD OR FOPEN_MODETEXT;      // Opens for reading in text format
				fbFileOpen.ePath := PATH_GENERIC;
				fbFileOpen.tTimeout := T#30S;
				fbFileOpen(bExecute:= FALSE);
				fbFileOpen(bExecute:= TRUE);
				
				// wait until fail isopened
				udiWaitFileOpenCycles := 0;
				 stStatemachine.uinState_old := stStatemachine.uinState;
			END_IF
			
			fbFileOpen(bExecute:= TRUE);
			
			IF ((fbFileOpen.bError=FALSE) AND ((fbFileOpen.bBusy) OR (fbFileOpen.hFile=0))) THEN
				udiWaitFileOpenCycles := udiWaitFileOpenCycles + 1;	
			ELSE
				IF (fbFileOpen.bError=TRUE) THEN
					// file not found
					IF (fbFileOpen.nErrId=16#70C) THEN
						strInfo := CONCAT(STR1:='template/config file: not found: ',STR2:= In_strPath); 
						strInfo := CONCAT(STR1:=strInfo,STR2:= In_strCfgFileName); 
						Out_udiStatus := fbFileOpen.nErrId;
						RETURN;
					ELSE 
						strInfo := CONCAT(STR1:='template/config file: no more free file handles / unknown or invalid nMode or ePath parameter: ',STR2:= In_strPath); 
						strInfo := CONCAT(STR1:=strInfo,STR2:= In_strCfgFileName); 
						Out_udiStatus := fbFileOpen.nErrId;
						RETURN;
					END_IF
				ELSE
					stStatemachine.uinState := 3;
				END_IF
			END_IF
		
		3:	// read config file in temp buffer allocate buffer
			// Entry action
			IF (stStatemachine.uinState_old <> stStatemachine.uinState) THEN
				//*********************************************************
				// read template file
				fbFileRead.sNetId:=''; // local file access
				fbFileRead.hFile:=fbFileOpen.hFile;
				fbFileRead.tTimeout:=T#3S;
				// create buffer
				fbFileRead.pReadBuff := M_AllocMEM(uinFileSize);
				pDelReadPointer := fbFileRead.pReadBuff; // pointer for release
				fbFileRead.cbReadLen := uinFileSize;
				
				IF (fbFileRead.pReadBuff=TC3_MEMMAN.NULL) THEN
					strInfo := CONCAT(STR1:='template/config file: alloc file buffer invalid: ',STR2:= In_strPath);
					strInfo := CONCAT(STR1:=strInfo,STR2:= In_strCfgFileName);
					Out_udiStatus := FileLc.cERR_ALLOC_BUFFER_FILE_CONFIG;
					RETURN;
				END_IF
				
				//valid buffer allocated
				fbFileRead(bExecute:=FALSE);
				fbFileRead(bExecute:=TRUE);
				udiWaitFileReadCycles := 0;
					
				 stStatemachine.uinState_old := stStatemachine.uinState;
			END_IF
			
			fbFileRead();	
			
			// read file binary
			IF (fbFileRead.bBusy) THEN
				udiWaitFileReadCycles := udiWaitFileReadCycles + 1;
			ELSE
				
			//test variabel
		MEMSET(destAddr:=pstrTmp,fillByte:=0,n:= SIZEOF(strTmp));
		MEMCPY(destAddr:=pstrTmp,srcAddr:=fbFileRead.pReadBuff,n:= (SIZEOF(strTmp)-1)); // zero determining string
		
				IF (fbFileRead.bError=FALSE) THEN
					IF (fbFileRead.cbRead<UINT_TO_UDINT(uinFileSize)) THEN // enough memory for whole cfg file allocated
						// allocated buffer is ok
						udiFileConfigLen := fbFileRead.cbRead; // file len read
						stStatemachine.uinState := stStatemachine.uinState  + 1;
					ELSE
						// buffer size to small! 
						
						// reset file read pointer
						fbFileSeek.sNetId:=''; // local file access
						fbFileSeek.hFile:=fbFileOpen.hFile;
						fbFileSeek.eOrigin:=E_SeekOrigin.SEEK_SET; // start pos at beginning of file
						fbFileSeek.tTimeout:=T#3S;
						fbFileSeek.nSeekPos := 0; // at beginn of file
						fbFileSeek(bExecute:=FALSE);
						fbFileSeek(bExecute:=TRUE);
						WHILE (fbFileSeek.bBusy) DO
							udiWaitFileReadCycles := udiWaitFileReadCycles + 1;
							fbFileSeek(bExecute:=TRUE);
						END_WHILE
						
						//release old buffer
						__DELETE(pDelReadPointer);

						uinFileSize := LREAL_TO_UINT(UINT_TO_LREAL(uinFileSize) * 1.5); // create bigger buffer for next try
						
						stStatemachine.uinState_old := 0; // entry action alloc new buffer
					END_IF
					
				ELSE
					// error read file
					strInfo := CONCAT(STR1:='template/config file: error reading file: ',STR2:= In_strPath);
					strInfo := CONCAT(STR1:=strInfo,STR2:= In_strCfgFileName);
					Out_udiStatus := fbFileRead.nErrId;
					RETURN;
				END_IF;
			END_IF
				
			
			
		4:
			//*********************************************************	
			// parse template file
			// <TEMPLATE>pBuffer
			p_bytTemplateBegin := strstr(In_pStr:=fbFileRead.pReadBuff,In_pStrSearch:=ADR(FileLc.cTAG_TEMPLATE_B),In_bolAddStrSearchLen:= TRUE);
			p_bytTemplateEnd := strstr(In_pStr:=fbFileRead.pReadBuff,In_pStrSearch:=ADR(FileLc.cTAG_TEMPLATE_E),In_bolAddStrSearchLen:= FALSE);
			IF ((p_bytTemplateBegin=TC3_MEMMAN.NULL) OR (p_bytTemplateEnd=TC3_MEMMAN.NULL) OR (p_bytTemplateBegin>p_bytTemplateEnd)) THEN
				strInfo := CONCAT(STR1:='template/config file: parse error: ',STR2:= FileLc.cTAG_TEMPLATE_B);
				Out_udiStatus := FileLc.cERR_TEMPLATE_TAG;
				RETURN;
			END_IF
			
			// <CONFIG>
			p_bytConfigBegin := strstr(In_pStr:=fbFileRead.pReadBuff,In_pStrSearch:=ADR(FileLc.cTAG_CONFIG_B),In_bolAddStrSearchLen:= TRUE);
			p_bytConfigEnd := strstr(In_pStr:=fbFileRead.pReadBuff,In_pStrSearch:=ADR(FileLc.cTAG_CONFIG_E),In_bolAddStrSearchLen:= FALSE);
		
			IF ((p_bytConfigBegin=TC3_MEMMAN.NULL) OR (p_bytConfigEnd=TC3_MEMMAN.NULL) OR (p_bytConfigBegin>p_bytConfigEnd)) THEN
				strInfo := CONCAT(STR1:='template/config file: parse error: ',STR2:= FileLc.cTAG_CONFIG_B);
				Out_udiStatus := FileLc.cERR_CONFIG_TAG;
				RETURN;
			END_IF
			
			// <HEADER>
			p_bytHeaderBegin := strstr(In_pStr:=fbFileRead.pReadBuff,In_pStrSearch:=ADR(FileLc.cTAG_HEADER_B),In_bolAddStrSearchLen:= TRUE);
			p_bytHeaderEnd := strstr(In_pStr:=fbFileRead.pReadBuff,In_pStrSearch:=ADR(FileLc.cTAG_HEADER_E),In_bolAddStrSearchLen:= FALSE);
			IF ((p_bytHeaderBegin=TC3_MEMMAN.NULL) OR (p_bytHeaderEnd=TC3_MEMMAN.NULL) OR (p_bytHeaderBegin>p_bytHeaderEnd)) THEN
				strInfo := CONCAT(STR1:='template/config file: parse error: ',STR2:= FileLc.cTAG_HEADER_B);
				Out_udiStatus := FileLc.cERR_HEADER_TAG;
				RETURN;
			END_IF
			
			// <FOOTER>
			p_bytFooterBegin := strstr(In_pStr:=fbFileRead.pReadBuff,In_pStrSearch:=ADR(FileLc.cTAG_FOOTER_B),In_bolAddStrSearchLen:= TRUE);
			p_bytFooterEnd := strstr(In_pStr:=fbFileRead.pReadBuff,In_pStrSearch:=ADR(FileLc.cTAG_FOOTER_E),In_bolAddStrSearchLen:= FALSE);
			IF ((p_bytFooterBegin=TC3_MEMMAN.NULL) OR (p_bytFooterEnd=TC3_MEMMAN.NULL) OR (p_bytFooterBegin>p_bytFooterEnd)) THEN
				strInfo := CONCAT(STR1:='template/config file: parse error: ',STR2:= FileLc.cTAG_FOOTER_B);
				Out_udiStatus := FileLc.cERR_FOOTER_TAG;
				RETURN;
			END_IF
			
			// <RECORD>
			p_bytRecordBegin := strstr(In_pStr:=fbFileRead.pReadBuff,In_pStrSearch:=ADR(FileLc.cTAG_RECORD_B),In_bolAddStrSearchLen:= TRUE);
			p_bytRecordEnd := strstr(In_pStr:=fbFileRead.pReadBuff,In_pStrSearch:=ADR(FileLc.cTAG_RECORD_E),In_bolAddStrSearchLen:= FALSE);
			IF ((p_bytRecordBegin=TC3_MEMMAN.NULL) OR (p_bytRecordEnd=TC3_MEMMAN.NULL) OR (p_bytRecordBegin>p_bytRecordEnd)) THEN
				strInfo := CONCAT(STR1:='template/config file: parse error: ',STR2:= FileLc.cTAG_RECORD_B);
				Out_udiStatus := FileLc.cERR_RECORD_TAG;
				RETURN;
			END_IF
			
			//*********************************************************	
			// check header
			// allocate memory for header text
			uinTmpLen := UDINT_TO_UINT(p_bytHeaderEnd-p_bytHeaderBegin); // with key words -> len > necessary...
		//test variabel
			MEMSET(destAddr:=pstrTmp,fillByte:=0,n:= SIZEOF(strTmp));
			MEMCPY(destAddr:=pstrTmp,srcAddr:=p_bytHeaderBegin,n:= (SIZEOF(strTmp)-1)); // zero determining string
			
			
			In_pstSysInfo^.p_bytHeaderText := M_AllocMEM(uinTmpLen);
			IF (In_pstSysInfo^.p_bytHeaderText=TC3_MEMMAN.NULL) THEN
				strInfo := 'template/config file: alloc memory for header text failed';
				Out_udiStatus := FileLc.cERR_ALLOC_MEMORY;
				RETURN;
			END_IF
			p_bytTmpDestAdr := In_pstSysInfo^.p_bytHeaderText;
			p_bytTmpSrcAdr := p_bytHeaderBegin;
			uinTmpLen := 0;
			REPEAT
				p_bytRowBegin := strstr(In_pStr:=p_bytTmpSrcAdr,In_pStrSearch:=ADR(FileLc.cTAG_ROW_B),In_bolAddStrSearchLen:= TRUE);
				p_bytRowEnd := strstr(In_pStr:=p_bytTmpSrcAdr,In_pStrSearch:=ADR(FileLc.cTAG_ROW_E),In_bolAddStrSearchLen:= FALSE);
				IF ((p_bytRowBegin<>TC3_MEMMAN.NULL) AND (p_bytRowEnd<>TC3_MEMMAN.NULL) 
					AND (p_bytRowBegin<p_bytHeaderEnd) AND (p_bytRowEnd<p_bytHeaderEnd)) THEN
					IF (p_bytRowBegin>p_bytRowEnd) THEN
						strInfo := CONCAT(STR1:='template/config file: parse error: ',STR2:= FileLc.cTAG_ROW_B);
						strInfo := CONCAT(STR1:=strInfo,STR2:= ' in :');
						strInfo := CONCAT(STR1:=strInfo,STR2:= FileLc.cTAG_HEADER_B);
						Out_udiStatus := FileLc.cERR_ROW_TAG;
						RETURN;
					END_IF
					uinTmpLen := uinTmpLen + DWORD_TO_UINT(p_bytRowEnd-p_bytRowBegin);
					MEMCPY(destAddr:=p_bytTmpDestAdr,srcAddr:=p_bytRowBegin,n:=(p_bytRowEnd-p_bytRowBegin)); // copy row section
			//test variabel
			MEMSET(destAddr:=pstrTmp,fillByte:=0,n:= SIZEOF(strTmp));
			MEMCPY(destAddr:=pstrTmp,srcAddr:=p_bytTmpDestAdr,n:= (SIZEOF(strTmp)-1)); // zero determining string
			
					p_bytTmpDestAdr := p_bytTmpDestAdr + p_bytRowEnd - p_bytRowBegin; //calculate next adress to add texts
					uinTmpLen := uinTmpLen + SIZEOF(FileLc.cEOL);
					MEMCPY(destAddr:=p_bytTmpDestAdr,srcAddr:=ADR(FileLc.cEOL),n:=SIZEOF(FileLc.cEOL)); //add end of line
					p_bytTmpDestAdr := p_bytTmpDestAdr + SIZEOF(FileLc.cEOL);
					p_bytTmpSrcAdr := p_bytRowEnd + Tc2_Standard.LEN(STR:=FileLc.cTAG_ROW_E);
				ELSE
					p_bytRowBegin := TC3_MEMMAN.NULL;
				END_IF
			UNTIL(p_bytRowBegin=TC3_MEMMAN.NULL)
			END_REPEAT
			In_pstSysInfo^.udiHeaderTextLen := UINT_TO_UDINT(uinTmpLen);
			
			
			//*********************************************************	
			// check footer
			// allocate memory for footer text
			uinTmpLen := UDINT_TO_UINT(p_bytFooterEnd-p_bytFooterBegin);// with key words -> len > necessary...
			
			In_pstSysInfo^.p_bytFooterText := M_AllocMEM(uinTmpLen);
			IF (In_pstSysInfo^.p_bytFooterText=TC3_MEMMAN.NULL) THEN
				strInfo := 'template/config file: alloc memory for footer text failed';
				Out_udiStatus := FileLc.cERR_ALLOC_MEMORY;
				RETURN;
			END_IF
			p_bytTmpDestAdr := In_pstSysInfo^.p_bytFooterText;
			p_bytTmpSrcAdr := p_bytFooterBegin;
			uinTmpLen := 0;
			REPEAT
				p_bytRowBegin := strstr(In_pStr:=p_bytTmpSrcAdr,In_pStrSearch:=ADR(FileLc.cTAG_ROW_B),In_bolAddStrSearchLen:= TRUE);
				p_bytRowEnd := strstr(In_pStr:=p_bytTmpSrcAdr,In_pStrSearch:=ADR(FileLc.cTAG_ROW_E),In_bolAddStrSearchLen:= FALSE);
				IF ((p_bytRowBegin<>TC3_MEMMAN.NULL) AND (p_bytRowEnd<>TC3_MEMMAN.NULL) 
					AND (p_bytRowBegin<p_bytFooterEnd) AND (p_bytRowEnd<p_bytFooterEnd)) THEN
					IF (p_bytRowBegin>p_bytRowEnd) THEN
						strInfo := CONCAT(STR1:='template/config file: parse error: ',STR2:= FileLc.cTAG_ROW_B);
						strInfo := CONCAT(STR1:=strInfo,STR2:= ' in :');
						strInfo := CONCAT(STR1:=strInfo,STR2:= FileLc.cTAG_FOOTER_B);
						Out_udiStatus := FileLc.cERR_ROW_TAG;
						RETURN;
					END_IF
					uinTmpLen := uinTmpLen + DWORD_TO_UINT(p_bytRowEnd-p_bytRowBegin);
					MEMCPY(destAddr:=p_bytTmpDestAdr,srcAddr:=p_bytRowBegin,n:=(p_bytRowEnd-p_bytRowBegin)); // copy row section
					p_bytTmpDestAdr := p_bytTmpDestAdr + p_bytRowEnd - p_bytRowBegin; //calculate next adress to add texts
					uinTmpLen := uinTmpLen + SIZEOF(FileLc.cEOL);
					MEMCPY(destAddr:=p_bytTmpDestAdr,srcAddr:=ADR(FileLc.cEOL),n:=SIZEOF(FileLc.cEOL)); //add end of line
					p_bytTmpDestAdr := p_bytTmpDestAdr + SIZEOF(FileLc.cEOL);
					p_bytTmpSrcAdr := p_bytRowEnd + Tc2_Standard.LEN(STR:=FileLc.cTAG_ROW_E);
				ELSE
					p_bytRowBegin := TC3_MEMMAN.NULL;
				END_IF
			UNTIL(p_bytRowBegin=TC3_MEMMAN.NULL)
			END_REPEAT
			In_pstSysInfo^.udiFooterTextLen := UINT_TO_UDINT(uinTmpLen);
			
			//*********************************************************	
			// check RECORD
			uinItemCount := 0;
			p_bytTmpSrcAdr := p_bytRecordBegin;
			
			// count all items in record tag
			REPEAT
				p_bytItemBegin := strstr(In_pStr:=p_bytTmpSrcAdr,In_pStrSearch:=ADR(FileLc.cTAG_ITEM_B),In_bolAddStrSearchLen:= TRUE);
				p_bytItemEnd := strstr(In_pStr:=p_bytTmpSrcAdr,In_pStrSearch:=ADR(FileLc.cTAG_ITEM_E),In_bolAddStrSearchLen:= FALSE);
				
				IF ((p_bytItemBegin<>TC3_MEMMAN.NULL) AND (p_bytItemEnd<>TC3_MEMMAN.NULL) 
					AND (p_bytItemBegin<p_bytRecordEnd) AND (p_bytItemEnd<p_bytRecordEnd)) THEN
					p_bytTmpSrcAdr := p_bytItemEnd + LEN(STR:=FileLc.cTAG_ITEM_E); 
					
					// plausibility check
					IF (p_bytItemBegin>p_bytItemEnd) THEN
						strInfo := CONCAT(STR1:='template/config file: parse error: ',STR2:= FileLc.cTAG_ITEM_B);
						strInfo := CONCAT(STR1:=strInfo,STR2:= ' in :');
						strInfo := CONCAT(STR1:=strInfo,STR2:= FileLc.cTAG_RECORD_B);
						Out_udiStatus := FileLc.cERR_ITEM_TAG;
						RETURN;
					END_IF
					// item tag count
					uinItemCount := uinItemCount +1;
				ELSE
					p_bytItemBegin := TC3_MEMMAN.NULL;
				END_IF
				
			UNTIL(p_bytItemBegin=TC3_MEMMAN.NULL)
			END_REPEAT
			
			// save found number of items
			In_pstSysInfo^.stItemInfo.uinActNbrOfItems := uinItemCount;
			
			// allocate memory for ItemData list
			FOR ii:=0 TO Queue.cMAX_NR_OF_TASKS BY 1 DO
				In_pstSysInfo^.stItemInfo.a_p_bytItemDataList[ii] := M_AllocMEM(uinItemCount*SIZEOF(T_FileLc_ItemData));
				IF (In_pstSysInfo^.stItemInfo.a_p_bytItemDataList[ii]=TC3_MEMMAN.NULL) THEN
					strInfo := 'template/config file: alloc memory for item data list failed';
					Out_udiStatus := FileLc.cERR_ALLOC_MEMORY;
					RETURN;
				END_IF
			END_FOR
			stStatemachine.uinState := stStatemachine.uinState  + 1;
		
		5:
			// allocate memory for ItemCfg list
			In_pstSysInfo^.stItemInfo.p_bytItemCfgList := M_AllocMEM(uinItemCount*SIZEOF(T_FileLc_ItemCfg));
			IF (In_pstSysInfo^.stItemInfo.p_bytItemCfgList=TC3_MEMMAN.NULL) THEN
				strInfo := 'template/config file: alloc memory for item config list failed';
				Out_udiStatus := FileLc.cERR_ALLOC_MEMORY;
				RETURN;
			END_IF
			p_stItemCfgList := In_pstSysInfo^.stItemInfo.p_bytItemCfgList;
			
			//*********************************************************	
			// in RECORD, search all item-tags
			uinItemCount := 0;
			p_bytTmpSrcAdr := p_bytRecordBegin;
			
			// count all items in record tag
			REPEAT
				p_bytItemBegin := strstr(In_pStr:=p_bytTmpSrcAdr,In_pStrSearch:=ADR(FileLc.cTAG_ITEM_B),In_bolAddStrSearchLen:= TRUE);
				p_bytItemEnd := strstr(In_pStr:=p_bytTmpSrcAdr,In_pStrSearch:=ADR(FileLc.cTAG_ITEM_E),In_bolAddStrSearchLen:= FALSE);
				
				IF ((p_bytItemBegin<>TC3_MEMMAN.NULL) AND (p_bytItemEnd<>TC3_MEMMAN.NULL) 
					AND (p_bytItemBegin<p_bytRecordEnd) AND (p_bytItemEnd<p_bytRecordEnd)) THEN
					
					// plausibility check
					IF (p_bytItemBegin>p_bytItemEnd) THEN
						strInfo := CONCAT(STR1:='template/config file: parse error: ',STR2:= FileLc.cTAG_ITEM_B);
						strInfo := CONCAT(STR1:=strInfo,STR2:= ' in :');
						strInfo := CONCAT(STR1:=strInfo,STR2:= FileLc.cTAG_RECORD_B);
						Out_udiStatus := FileLc.cERR_ITEM_TAG;
						RETURN;
					END_IF
					//test variabel
		MEMSET(destAddr:=pstrTmp,fillByte:=0,n:= SIZEOF(strTmp));
		MEMCPY(destAddr:=pstrTmp,srcAddr:=p_bytItemBegin,n:= (SIZEOF(strTmp)-1)); // zero determining string
		
					p_bytTmpSrcAdr := p_bytItemEnd + LEN(STR:=FileLc.cTAG_ITEM_E);
					udiTmpLen := p_bytItemEnd-p_bytItemBegin;
					IF (MEMCMP(pBuf1:=p_bytItemBegin,pBuf2:=ADR(FileLc.cITEM_UNIX_DATE_TIME),udiTmpLen) = 0) THEN
						p_stItemCfgList[uinItemCount].dinPvId := FileLc.cPVTYPE_UNIX_DATE_TIME;		
					ELSIF(MEMCMP(pBuf1:=p_bytItemBegin,pBuf2:=ADR(FileLc.cITEM_UNIX_DATE_TIME_STR),udiTmpLen) = 0) THEN
						p_stItemCfgList[uinItemCount].dinPvId := FileLc.cPVTYPE_UNIX_DATE_TIME_STR;	
					ELSIF(MEMCMP(pBuf1:=p_bytItemBegin,pBuf2:=ADR(FileLc.cITEM_EXCEL_DATE_TIME),udiTmpLen) = 0) THEN
						p_stItemCfgList[uinItemCount].dinPvId := FileLc.cPVTYPE_EXCEL_DATE_TIME;	
					ELSIF(MEMCMP(pBuf1:=p_bytItemBegin,pBuf2:=ADR(FileLc.cITEM_DATE_SLASH_TIME_COLON),udiTmpLen) = 0) THEN
						p_stItemCfgList[uinItemCount].dinPvId := FileLc.cPVTYPE_DATE_SLASH_TIME_COLON;		
					ELSIF(MEMCMP(pBuf1:=p_bytItemBegin,pBuf2:=ADR(FileLc.cITEM_TIME_MILLI),udiTmpLen) = 0) THEN
						p_stItemCfgList[uinItemCount].dinPvId := FileLc.cPVTYPE_TIME_MILLI;	
					ELSIF(MEMCMP(pBuf1:=p_bytItemBegin,pBuf2:=ADR(FileLc.cITEM_BL_LOGTYP),udiTmpLen) = 0) THEN
						p_stItemCfgList[uinItemCount].dinPvId := FileLc.cPVTYPE_BL_LOGTYP;	
					ELSIF(MEMCMP(pBuf1:=p_bytItemBegin,pBuf2:=ADR(FileLc.cITEM_BL_CTRL_ID),udiTmpLen) = 0) THEN
						p_stItemCfgList[uinItemCount].dinPvId := FileLc.cPVTYPE_BL_CTRL_ID;	
					ELSIF(MEMCMP(pBuf1:=p_bytItemBegin,pBuf2:=ADR(FileLc.cITEM_BL_STRING1),udiTmpLen) = 0) THEN
						p_stItemCfgList[uinItemCount].dinPvId := FileLc.cPVTYPE_BL_STRING1;	
					ELSIF(MEMCMP(pBuf1:=p_bytItemBegin,pBuf2:=ADR(FileLc.cITEM_BL_STRING2),udiTmpLen) = 0) THEN
						p_stItemCfgList[uinItemCount].dinPvId := FileLc.cPVTYPE_BL_STRING2;	
					ELSIF(MEMCMP(pBuf1:=p_bytItemBegin,pBuf2:=ADR(FileLc.cITEM_BL_PAR1),udiTmpLen) = 0) THEN
						p_stItemCfgList[uinItemCount].dinPvId := FileLc.cPVTYPE_BL_PAR1;	
					ELSIF(MEMCMP(pBuf1:=p_bytItemBegin,pBuf2:=ADR(FileLc.cITEM_BL_PAR2),udiTmpLen) = 0) THEN
						p_stItemCfgList[uinItemCount].dinPvId := FileLc.cPVTYPE_BL_PAR2;
					ELSIF(MEMCMP(pBuf1:=p_bytItemBegin,pBuf2:=ADR(FileLc.cITEM_BL_PAR3),udiTmpLen) = 0) THEN
						p_stItemCfgList[uinItemCount].dinPvId := FileLc.cPVTYPE_BL_PAR3;
					ELSIF(MEMCMP(pBuf1:=p_bytItemBegin,pBuf2:=ADR(FileLc.cITEM_BL_PAR4),udiTmpLen) = 0) THEN
						p_stItemCfgList[uinItemCount].dinPvId := FileLc.cPVTYPE_BL_PAR4;
					ELSE
						MEMSET(destAddr := ADR(strTmp),0,SIZEOF(strTmp));
						IF (udiTmpLen < SIZEOF(strTmp)) THEN
							MEMCPY(destAddr := ADR(strTmp),srcAddr := p_bytItemBegin,udiTmpLen);
							p_stItemCfgList[uinItemCount].dinPvId := STRING_TO_DINT(strTmp);
						ELSE
							strInfo := CONCAT(STR1:='template/config file: parse error item definition larger than defined string: ',STR2:= FileLc.cTAG_ITEM_B);
							strInfo := CONCAT(STR1:=strInfo,STR2:= ' in :');
							strInfo := CONCAT(STR1:=strInfo,STR2:= FileLc.cTAG_RECORD_B);
							Out_udiStatus := FileLc.cERR_ITEM_TAG;
							RETURN;
						END_IF
					END_IF
					
					IF (uinItemCount=0) THEN // only for the first element
						// PreText
						udiTmpLen := p_bytItemBegin-Tc2_Standard.LEN(STR:=FileLc.cTAG_ITEM_B)-p_bytRecordBegin;
						IF (udiTmpLen>FileLc.cPRE_POST_TEXTLEN) THEN
							udiTmpLen := FileLc.cPRE_POST_TEXTLEN - 1; //-1 -> strEnd!
						END_IF
						MEMSET(destAddr := ADR(In_pstSysInfo^.stItemInfo.strPreItemText),0,SIZEOF(In_pstSysInfo^.stItemInfo.strPreItemText));
						MEMCPY(destAddr:=ADR(In_pstSysInfo^.stItemInfo.strPreItemText), p_bytRecordBegin, udiTmpLen);
					ELSE
						// Post item text
						udiTmpLen := p_bytItemBegin-Tc2_Standard.LEN(STR:=FileLc.cTAG_ITEM_B)-p_bytLastPos;
						IF (udiTmpLen>FileLc.cPRE_POST_TEXTLEN) THEN
							udiTmpLen := FileLc.cPRE_POST_TEXTLEN - 1; //-1 -> strEnd!
						END_IF
						MEMSET(destAddr := ADR(p_stItemCfgList[uinItemCount-1].strPostText),0,SIZEOF(p_stItemCfgList[uinItemCount-1].strPostText));
						MEMCPY(destAddr:=ADR(p_stItemCfgList[uinItemCount-1].strPostText), p_bytLastPos, udiTmpLen);
					END_IF
					
					// save last position of ITEM entry
					p_bytLastPos := p_bytItemEnd + Tc2_Standard.LEN(STR:=FileLc.cTAG_ITEM_E);
					// item tag count
					uinItemCount := uinItemCount +1;
				ELSE
					p_bytItemBegin := TC3_MEMMAN.NULL;
				END_IF
				
			UNTIL(p_bytItemBegin=TC3_MEMMAN.NULL)
			END_REPEAT
			
			// manage last element
			udiTmpLen := p_bytRecordEnd-p_bytLastPos;
			IF (udiTmpLen>FileLc.cPRE_POST_TEXTLEN) THEN
				udiTmpLen := FileLc.cPRE_POST_TEXTLEN - 1; //-1 -> strEnd!
			END_IF
			MEMCPY(destAddr:=ADR(p_stItemCfgList[uinItemCount-1].strPostText), p_bytLastPos, udiTmpLen);
			
			//*********************************************************	
			// check CONFIG 
			
			//**** <LOGFILE_PRAEFIX>
			p_bytConfigValBegin := strstr(In_pStr:=p_bytConfigBegin,In_pStrSearch:=ADR(FileLc.cTAG_CFG_LOGFILE_PRAEFIX_B),In_bolAddStrSearchLen:= TRUE);
			p_bytConfigValEnd := strstr(In_pStr:=p_bytConfigBegin,In_pStrSearch:=ADR(FileLc.cTAG_CFG_LOGFILE_PRAEFIX_E),In_bolAddStrSearchLen:= FALSE);
			IF ((p_bytConfigValBegin<>TC3_MEMMAN.NULL) AND (p_bytConfigValEnd<>TC3_MEMMAN.NULL) AND (p_bytConfigValBegin<p_bytConfigValEnd) AND (p_bytConfigValEnd<p_bytConfigEnd)) THEN
				MEMSET(destAddr := ADR(strTmp),0,SIZEOF(strTmp));
				udiTmpLen := p_bytConfigValEnd - p_bytConfigValBegin;
		
				IF (SIZEOF(strTmp)>udiTmpLen) THEN
					MEMCPY(destAddr := ADR(strTmp),srcAddr := p_bytConfigValBegin,udiTmpLen);	
				ELSE
					strTmp := FileLc.cCFG_LOGFILE_NAME; // error - load default
				END_IF
			ELSE
				strTmp := FileLc.cCFG_LOGFILE_NAME; // error - load default
			END_IF
			In_pstSysInfo^.stConfig.strLogFileNamePraeFix := strTmp;
			
			//**** <LOGFILE_EXT>
			p_bytConfigValBegin := strstr(In_pStr:=p_bytConfigBegin,In_pStrSearch:=ADR(FileLc.cTAG_CFG_LOGFILE_EXT_B),In_bolAddStrSearchLen:= TRUE);
			p_bytConfigValEnd := strstr(In_pStr:=p_bytConfigBegin,In_pStrSearch:=ADR(FileLc.cTAG_CFG_LOGFILE_EXT_E),In_bolAddStrSearchLen:= FALSE);
			IF ((p_bytConfigValBegin<>TC3_MEMMAN.NULL) AND (p_bytConfigValEnd<>TC3_MEMMAN.NULL) AND (p_bytConfigValBegin<p_bytConfigValEnd) AND (p_bytConfigValEnd<p_bytConfigEnd)) THEN
				MEMSET(destAddr := ADR(strTmp),0,SIZEOF(strTmp));
				udiTmpLen := p_bytConfigValEnd - p_bytConfigValBegin;
		
				IF (SIZEOF(strTmp)>udiTmpLen) THEN
					MEMCPY(destAddr := ADR(strTmp),srcAddr := p_bytConfigValBegin,udiTmpLen);	
				ELSE
					strTmp := FileLc.cCFG_LOGFILE_EXT; // error - load default
				END_IF
			ELSE
				strTmp := FileLc.cCFG_LOGFILE_EXT; // error - load default
			END_IF
			In_pstSysInfo^.stConfig.strLogFileNameExt := strTmp;
			
			//**** <LOG_TIMESTAMP>
			
			p_bytConfigValBegin := strstr(In_pStr:=p_bytConfigBegin,In_pStrSearch:=ADR(FileLc.cTAG_CFG_LOG_TIMESTAMP_B),In_bolAddStrSearchLen:= TRUE);
			p_bytConfigValEnd := strstr(In_pStr:=p_bytConfigBegin,In_pStrSearch:=ADR(FileLc.cTAG_CFG_LOG_TIMESTAMP_E),In_bolAddStrSearchLen:= FALSE);
			IF ((p_bytConfigValBegin<>TC3_MEMMAN.NULL) AND (p_bytConfigValEnd<>TC3_MEMMAN.NULL) AND (p_bytConfigValBegin<p_bytConfigValEnd) AND (p_bytConfigValEnd<p_bytConfigEnd)) THEN
				MEMSET(destAddr := ADR(strTmp),0,SIZEOF(strTmp));
				udiTmpLen := p_bytConfigValEnd - p_bytConfigValBegin;
		
				IF (SIZEOF(strTmp)>udiTmpLen) THEN
					MEMCPY(destAddr := ADR(strTmp),srcAddr := p_bytConfigValBegin,udiTmpLen);	
					IF (FIND(STR1:=strTmp,STR2:=FileLc.cLOG_TIMESTAMP_WIN)<>0)THEN // win defiend
						bolTmp := TRUE;
					ELSE
						bolTmp := FALSE;
					END_IF
				ELSE
					bolTmp := FALSE; // error - load default - local drive access
				END_IF
			ELSE
				bolTmp := FALSE; // error - load default - local drive access
			END_IF
			In_pstSysInfo^.stConfig.bolUseLocalTimeStamp := bolTmp;
			
			//**** <LOGFILE_SNETID>
			p_bytConfigValBegin := strstr(In_pStr:=p_bytConfigBegin,In_pStrSearch:=ADR(FileLc.cTAG_CFG_LOGFILE_SNETID_B),In_bolAddStrSearchLen:= TRUE);
			p_bytConfigValEnd := strstr(In_pStr:=p_bytConfigBegin,In_pStrSearch:=ADR(FileLc.cTAG_CFG_LOGFILE_SNETID_E),In_bolAddStrSearchLen:= FALSE);
			IF ((p_bytConfigValBegin<>TC3_MEMMAN.NULL) AND (p_bytConfigValEnd<>TC3_MEMMAN.NULL) AND (p_bytConfigValBegin<p_bytConfigValEnd) AND (p_bytConfigValEnd<p_bytConfigEnd)) THEN
				MEMSET(destAddr := ADR(strTmp),0,SIZEOF(strTmp));
				udiTmpLen := p_bytConfigValEnd - p_bytConfigValBegin;
		
				IF (SIZEOF(strTmp)>udiTmpLen) THEN
					MEMCPY(destAddr := ADR(strTmp),srcAddr := p_bytConfigValBegin,udiTmpLen);	
				ELSE
					strTmp := ''; // error - load default - local drive access
				END_IF
			ELSE
				strTmp :=  ''; // error - load default - local drive access
			END_IF
			In_pstSysInfo^.stConfig.strLogNetId := strTmp;
			
			//**** <LOGFILE_PATH>
			p_bytConfigValBegin := strstr(In_pStr:=p_bytConfigBegin,In_pStrSearch:=ADR(FileLc.cTAG_CFG_LOGFILE_PATH_B),In_bolAddStrSearchLen:= TRUE);
			p_bytConfigValEnd := strstr(In_pStr:=p_bytConfigBegin,In_pStrSearch:=ADR(FileLc.cTAG_CFG_LOGFILE_PATH_E),In_bolAddStrSearchLen:= FALSE);
			IF ((p_bytConfigValBegin<>TC3_MEMMAN.NULL) AND (p_bytConfigValEnd<>TC3_MEMMAN.NULL) AND (p_bytConfigValBegin<p_bytConfigValEnd) AND (p_bytConfigValEnd<p_bytConfigEnd)) THEN
				MEMSET(destAddr := ADR(strTmp),0,SIZEOF(strTmp));
				udiTmpLen := p_bytConfigValEnd - p_bytConfigValBegin;
		
				IF (SIZEOF(strTmp)>udiTmpLen) THEN
					MEMCPY(destAddr := ADR(strTmp),srcAddr := p_bytConfigValBegin,udiTmpLen);	
				ELSE
					strTmp := In_strPath; // error - load default
				END_IF
			ELSE
				strTmp := In_strPath; // error - load default
			END_IF
			In_pstSysInfo^.stConfig.strLogPath := CONCAT(STR1:=strTmp ,STR2:= '\');
			
			//**** <QEUE_LEN>
			p_bytConfigValBegin := strstr(In_pStr:=p_bytConfigBegin,In_pStrSearch:=ADR(FileLc.cTAG_CFG_QUEUE_LEN_B),In_bolAddStrSearchLen:= TRUE);
			p_bytConfigValEnd := strstr(In_pStr:=p_bytConfigBegin,In_pStrSearch:=ADR(FileLc.cTAG_CFG_QUEUE_LEN_E),In_bolAddStrSearchLen:= FALSE);
			IF ((p_bytConfigValBegin<>TC3_MEMMAN.NULL) AND (p_bytConfigValEnd<>TC3_MEMMAN.NULL) AND (p_bytConfigValBegin<p_bytConfigValEnd) AND (p_bytConfigValEnd<p_bytConfigEnd)) THEN
				MEMSET(destAddr := ADR(strTmp),0,SIZEOF(strTmp));
				udiTmpLen := p_bytConfigValEnd - p_bytConfigValBegin;
		
				IF (SIZEOF(strTmp)>udiTmpLen) THEN
					MEMCPY(destAddr := ADR(strTmp),srcAddr := p_bytConfigValBegin,udiTmpLen);	
					In_pstSysInfo^.stConfig.udiQueueLen := STRING_TO_UDINT(strTmp);
				ELSE
					In_pstSysInfo^.stConfig.udiQueueLen := FileLc.cCFG_QUEUE_LEN; // error - load default
				END_IF
			ELSE
				In_pstSysInfo^.stConfig.udiQueueLen := FileLc.cCFG_QUEUE_LEN; // error - load default
			END_IF
			
			//**** <MASK>
			p_bytConfigValBegin := strstr(In_pStr:=p_bytConfigBegin,In_pStrSearch:=ADR(FileLc.cTAG_CFG_MASK_B),In_bolAddStrSearchLen:= TRUE);
			p_bytConfigValEnd := strstr(In_pStr:=p_bytConfigBegin,In_pStrSearch:=ADR(FileLc.cTAG_CFG_MASK_E),In_bolAddStrSearchLen:= FALSE);
			IF ((p_bytConfigValBegin<>TC3_MEMMAN.NULL) AND (p_bytConfigValEnd<>TC3_MEMMAN.NULL) AND (p_bytConfigValBegin<p_bytConfigValEnd) AND (p_bytConfigValEnd<p_bytConfigEnd)) THEN
				MEMSET(destAddr := ADR(strTmp),0,SIZEOF(strTmp));
				udiTmpLen := p_bytConfigValEnd - p_bytConfigValBegin;
		
				IF (SIZEOF(strTmp)>udiTmpLen) THEN
					MEMCPY(destAddr := ADR(strTmp),srcAddr := p_bytConfigValBegin,udiTmpLen);	
					In_pstSysInfo^.udiMask := STRING_TO_UDINT(strTmp);
				ELSE
					In_pstSysInfo^.udiMask := FileLc.cCFG_DEFAULT_MASK; // error - load default
				END_IF
			ELSE
				In_pstSysInfo^.udiMask := FileLc.cCFG_DEFAULT_MASK; // error - load default
			END_IF
			
			//**** <LOG_TYPE>
			p_bytConfigValBegin := strstr(In_pStr:=p_bytConfigBegin,In_pStrSearch:=ADR(FileLc.cTAG_CFG_LOGTYPE_B),In_bolAddStrSearchLen:= TRUE);
			p_bytConfigValEnd := strstr(In_pStr:=p_bytConfigBegin,In_pStrSearch:=ADR(FileLc.cTAG_CFG_LOGTYPE_E),In_bolAddStrSearchLen:= FALSE);
			IF ((p_bytConfigValBegin<>TC3_MEMMAN.NULL) AND (p_bytConfigValEnd<>TC3_MEMMAN.NULL) AND (p_bytConfigValBegin<p_bytConfigValEnd) AND (p_bytConfigValEnd<p_bytConfigEnd)) THEN
			
				udiTmpLen := p_bytConfigValEnd - p_bytConfigValBegin;	
				IF (MEMCMP(pBuf1:=p_bytConfigValBegin,pBuf2:=ADR(FileLc.cLOGTYP_BL_STR),n:=udiTmpLen)=0)THEN
					In_pstSysInfo^.uinLogTyp := FileLc.cLOGTYP_BL;
				ELSIF (MEMCMP(pBuf1:=p_bytConfigValBegin,pBuf2:=ADR(FileLc.cLOGTYP_PV_STR),n:=udiTmpLen)=0)THEN
					In_pstSysInfo^.uinLogTyp := FileLc.cLOGTYP_PV;
				ELSIF (MEMCMP(pBuf1:=p_bytConfigValBegin,pBuf2:=ADR(FileLc.cLOGTYP_DATA_STR),n:=udiTmpLen)=0)THEN
					In_pstSysInfo^.uinLogTyp := FileLc.cLOGTYP_DATA;
				ELSIF (MEMCMP(pBuf1:=p_bytConfigValBegin,pBuf2:=ADR(FileLc.cLOGTYP_OPEN_STR),n:=udiTmpLen)=0)THEN
					In_pstSysInfo^.uinLogTyp := FileLc.cLOGTYP_OPEN;	
				ELSE
					strInfo := CONCAT(STR1:='template/config file: parse error log typ not definde element: ',STR2:= FileLc.cTAG_CFG_LOGTYPE_B);
					Out_udiStatus := FileLc.cERR_INVALID_LOGTYP;
					RETURN;
				END_IF
			ELSE
				In_pstSysInfo^.uinLogTyp := FileLc.cLOGTYP_BL; // load default
			END_IF
			
			//**** <MAX_LOGFILES>
			p_bytConfigValBegin := strstr(In_pStr:=p_bytConfigBegin,In_pStrSearch:=ADR(FileLc.cTAG_CFG_MAX_LOGFILES_B),In_bolAddStrSearchLen:= TRUE);
			p_bytConfigValEnd := strstr(In_pStr:=p_bytConfigBegin,In_pStrSearch:=ADR(FileLc.cTAG_CFG_MAX_LOGFILES_E),In_bolAddStrSearchLen:= FALSE);
			IF ((p_bytConfigValBegin<>TC3_MEMMAN.NULL) AND (p_bytConfigValEnd<>TC3_MEMMAN.NULL) AND (p_bytConfigValBegin<p_bytConfigValEnd) AND (p_bytConfigValEnd<p_bytConfigEnd)) THEN
				MEMSET(destAddr := ADR(strTmp),0,SIZEOF(strTmp));
				udiTmpLen := p_bytConfigValEnd - p_bytConfigValBegin;
		
				IF (SIZEOF(strTmp)>udiTmpLen) THEN
					MEMCPY(destAddr := ADR(strTmp),srcAddr := p_bytConfigValBegin,udiTmpLen);	
					In_pstSysInfo^.stConfig.uinMaxNbrOfLogFiles := STRING_TO_UINT(strTmp);
				ELSE
					In_pstSysInfo^.stConfig.uinMaxNbrOfLogFiles := FileLc.cCFG_MAX_NBR_OF_LOGFILES; // error - load default
				END_IF
			ELSE
				In_pstSysInfo^.stConfig.uinMaxNbrOfLogFiles := FileLc.cCFG_MAX_NBR_OF_LOGFILES; // error - load default
			END_IF
			
			//**** <TIME_CHECK_MAX_FILE_NR>
			// max time check max file nr
			p_bytConfigValBegin := strstr(In_pStr:=p_bytConfigBegin,In_pStrSearch:=ADR(FileLc.cTAG_CFG_T_CHECK_MAX_FILE_NR_B),In_bolAddStrSearchLen:= TRUE);
			p_bytConfigValEnd := strstr(In_pStr:=p_bytConfigBegin,In_pStrSearch:=ADR(FileLc.cTAG_CFG_T_CHECK_MAX_FILE_NR_E),In_bolAddStrSearchLen:= FALSE);
			IF ((p_bytConfigValBegin<>TC3_MEMMAN.NULL) AND (p_bytConfigValEnd<>TC3_MEMMAN.NULL) AND (p_bytConfigValBegin<p_bytConfigValEnd) AND (p_bytConfigValEnd<p_bytConfigEnd)) THEN
				MEMSET(destAddr := ADR(strTmp),0,SIZEOF(strTmp));
				udiTmpLen := p_bytConfigValEnd - p_bytConfigValBegin;
		
				IF (SIZEOF(strTmp)>udiTmpLen) THEN
					MEMCPY(destAddr := ADR(strTmp),srcAddr := p_bytConfigValBegin,udiTmpLen);	
					In_pstSysInfo^.stConfig.udiTimeCheckMaxFileNr := STRING_TO_UDINT(strTmp)*1000; // defined in s -> ms
				ELSE
					In_pstSysInfo^.stConfig.udiTimeCheckMaxFileNr := FileLc.cTIME_CHECK_MAX_FILE_NR*1000; // defined in s -> ms// error - load default
				END_IF
			ELSE
				In_pstSysInfo^.stConfig.udiTimeCheckMaxFileNr:= FileLc.cTIME_CHECK_MAX_FILE_NR*1000; // defined in s -> ms// error - load default
			END_IF
			
			//**** <MAX_TIME_TO_WRITE>
			// max time between to file writes
			p_bytConfigValBegin := strstr(In_pStr:=p_bytConfigBegin,In_pStrSearch:=ADR(FileLc.cTAG_CFG_MAX_T_TO_WRITE_B),In_bolAddStrSearchLen:= TRUE);
			p_bytConfigValEnd := strstr(In_pStr:=p_bytConfigBegin,In_pStrSearch:=ADR(FileLc.cTAG_CFG_MAX_T_TO_WRITE_E),In_bolAddStrSearchLen:= FALSE);
			IF ((p_bytConfigValBegin<>TC3_MEMMAN.NULL) AND (p_bytConfigValEnd<>TC3_MEMMAN.NULL) AND (p_bytConfigValBegin<p_bytConfigValEnd) AND (p_bytConfigValEnd<p_bytConfigEnd)) THEN
				MEMSET(destAddr := ADR(strTmp),0,SIZEOF(strTmp));
				udiTmpLen := p_bytConfigValEnd - p_bytConfigValBegin;
		
				IF (SIZEOF(strTmp)>udiTmpLen) THEN
					MEMCPY(destAddr := ADR(strTmp),srcAddr := p_bytConfigValBegin,udiTmpLen);	
					In_pstSysInfo^.stConfig.udiMaxTimeWriteToFile := STRING_TO_UDINT(strTmp)*1000; // defined in s -> ms
				ELSE
					In_pstSysInfo^.stConfig.udiMaxTimeWriteToFile := FileLc.cCFG_TIME_WRITE_TO_FILE*1000; // defined in s -> ms// error - load default
				END_IF
			ELSE
				In_pstSysInfo^.stConfig.udiMaxTimeWriteToFile := FileLc.cCFG_TIME_WRITE_TO_FILE*1000; // defined in s -> ms// error - load default
			END_IF
			
			//**** <NEW_FILE_ON_RESTART>
			// >0 -> create always a new file on power up
			p_bytConfigValBegin := strstr(In_pStr:=p_bytConfigBegin,In_pStrSearch:=ADR(FileLc.cTAG_CFG_NEW_FILE_RESTART_B),In_bolAddStrSearchLen:= TRUE);
			p_bytConfigValEnd := strstr(In_pStr:=p_bytConfigBegin,In_pStrSearch:=ADR(FileLc.cTAG_CFG_NEW_FILE_RESTART_E),In_bolAddStrSearchLen:= FALSE);
			IF ((p_bytConfigValBegin<>TC3_MEMMAN.NULL) AND (p_bytConfigValEnd<>TC3_MEMMAN.NULL) AND (p_bytConfigValBegin<p_bytConfigValEnd) AND (p_bytConfigValEnd<p_bytConfigEnd)) THEN
				MEMSET(destAddr := ADR(strTmp),0,SIZEOF(strTmp));
				udiTmpLen := p_bytConfigValEnd - p_bytConfigValBegin;
		
				IF (SIZEOF(strTmp)>udiTmpLen) THEN
					MEMCPY(destAddr := ADR(strTmp),srcAddr := p_bytConfigValBegin,udiTmpLen);	
					In_pstSysInfo^.stConfig.uinNewFileOnRestart := STRING_TO_UINT(strTmp);
				ELSE
					In_pstSysInfo^.stConfig.uinNewFileOnRestart := 0; // error - load default
				END_IF
			ELSE
				In_pstSysInfo^.stConfig.uinNewFileOnRestart := 0; // error - load default
			END_IF
			
			//**** <MAX_ENTRIES_IN_FILE>
			// maximal number of entries in log file
			p_bytConfigValBegin := strstr(In_pStr:=p_bytConfigBegin,In_pStrSearch:=ADR(FileLc.cTAG_CFG_MAX_ENTR_IN_FILE_B),In_bolAddStrSearchLen:= TRUE);
			p_bytConfigValEnd := strstr(In_pStr:=p_bytConfigBegin,In_pStrSearch:=ADR(FileLc.cTAG_CFG_MAX_ENTR_IN_FILE_E),In_bolAddStrSearchLen:= FALSE);
			IF ((p_bytConfigValBegin<>TC3_MEMMAN.NULL) AND (p_bytConfigValEnd<>TC3_MEMMAN.NULL) AND (p_bytConfigValBegin<p_bytConfigValEnd) AND (p_bytConfigValEnd<p_bytConfigEnd)) THEN
				MEMSET(destAddr := ADR(strTmp),0,SIZEOF(strTmp));
				udiTmpLen := p_bytConfigValEnd - p_bytConfigValBegin;
		
				IF (SIZEOF(strTmp)>udiTmpLen) THEN
					MEMCPY(destAddr := ADR(strTmp),srcAddr := p_bytConfigValBegin,udiTmpLen);	
					In_pstSysInfo^.stConfig.udiMaxEntriesInFile := STRING_TO_UDINT(strTmp);
				ELSE
					In_pstSysInfo^.stConfig.udiMaxEntriesInFile := 0; // error - load default -> 0 no limit
				END_IF
			ELSE
				In_pstSysInfo^.stConfig.udiMaxEntriesInFile := 0; // error - load default -> 0 no limit
			END_IF
			
			//**** <MAX_FILE_SIZE_MB>
			// maximal size of a logfile [MBytes]
			p_bytConfigValBegin := strstr(In_pStr:=p_bytConfigBegin,In_pStrSearch:=ADR(FileLc.cTAG_CFG_MAX_FILE_SIZE_B),In_bolAddStrSearchLen:= TRUE);
			p_bytConfigValEnd := strstr(In_pStr:=p_bytConfigBegin,In_pStrSearch:=ADR(FileLc.cTAG_CFG_MAX_FILE_SIZE_E),In_bolAddStrSearchLen:= FALSE);
			IF ((p_bytConfigValBegin<>TC3_MEMMAN.NULL) AND (p_bytConfigValEnd<>TC3_MEMMAN.NULL) AND (p_bytConfigValBegin<p_bytConfigValEnd) AND (p_bytConfigValEnd<p_bytConfigEnd)) THEN
				MEMSET(destAddr := ADR(strTmp),0,SIZEOF(strTmp));
				udiTmpLen := p_bytConfigValEnd - p_bytConfigValBegin;
		
				IF (SIZEOF(strTmp)>udiTmpLen) THEN
					MEMCPY(destAddr := ADR(strTmp),srcAddr := p_bytConfigValBegin,udiTmpLen);	
					In_pstSysInfo^.stConfig.udiMaxFileSize := REAL_TO_UDINT(STRING_TO_REAL(strTmp)*1000000.0);// set in MB internal : bytes
				ELSE
					In_pstSysInfo^.stConfig.udiMaxFileSize := 0; // error - load default -> 0 no limit
				END_IF
			ELSE
				In_pstSysInfo^.stConfig.udiMaxFileSize := 0; // error - load default -> 0 no limit
			END_IF
			
			stStatemachine.uinState := stStatemachine.uinState  + 1;
		
		6:
			// Entry action
			IF (stStatemachine.uinState_old <> stStatemachine.uinState) THEN
				//*********************************************************
				// file close
				fbFileClose.sNetId := ''; // only local access
				fbFileClose.hFile := fbFileOpen.hFile; // only local access
				fbFileClose.tTimeout := T#3S;
				fbFileClose(bExecute:= FALSE);
				fbFileClose(bExecute:= TRUE);
				udiWaitFileCloseCycles := 0;
					
				 stStatemachine.uinState_old := stStatemachine.uinState;
			END_IF
				
			// wait UNTIL closed
			IF (fbFileClose.bBusy) THEN
				udiWaitFileCloseCycles := udiWaitFileCloseCycles + 1;
				fbFileClose(bExecute:=FALSE);
			ELSE
				IF fbFileClose.bError THEN
					strInfo := 'template/config file close failed';
					Out_udiStatus := fbFileClose.nErrId;
					RETURN;
				END_IF
				
				// delocate memory
				__DELETE(pDelReadPointer);
				
				// allocat for temporary item list
				// nbr of items * size for value output + nbf of items * Pre- and Post - Text
				// with this calculation is the buffer normally greater than necessary
				// cMAX_ITEM_CHAR has to be defined for worst case (big 4-byt values, date strings) so big
				udiTmpLen := (In_pstSysInfo^.stItemInfo.uinActNbrOfItems*FileLc.cMAX_ITEM_CHAR) + (In_pstSysInfo^.stItemInfo.uinActNbrOfItems*FileLc.cPRE_POST_TEXTLEN);
				In_pstSysInfo^.p_bytTmpRecordText := M_AllocMEM(In_SizeOfBuffer:=UDINT_TO_UINT(udiTmpLen));
				IF (In_pstSysInfo^.p_bytTmpRecordText=TC3_MEMMAN.NULL) THEN
					strInfo := 'template/config file: alloc memory for temp record text failed';
					Out_udiStatus := FileLc.cERR_ALLOC_MEMORY;
					RETURN;
				END_IF
				In_pstSysInfo^.udiTmpRecordSize := udiTmpLen;
				
				// allocat for temporary file buffer
				udiTmpLen := udiTmpLen*FileLc.cMAX_RECORDS_IN_FILE_BUF;
				In_pstSysInfo^.stFileHandler.p_bytTmpFileBuffer := M_AllocMEM(In_SizeOfBuffer:=UDINT_TO_UINT(udiTmpLen));
				IF (In_pstSysInfo^.stFileHandler.p_bytTmpFileBuffer=TC3_MEMMAN.NULL) THEN
					strInfo := 'template/config file: alloc memory for temp file buffer failed';
					Out_udiStatus := FileLc.cERR_ALLOC_MEMORY;
					RETURN;
				END_IF
				In_pstSysInfo^.stFileHandler.udiTmpFileBufferSize := udiTmpLen;
				stStatemachine.uinState := stStatemachine.uinState  + 1;
			END_IF
			
		
		7:
			stStatemachine.usiInitDone := 1;
			Out_bolDone := TRUE;
			strInfo := 'template/config file: successfully parsed';
			Out_udiStatus := 0;
	END_CASE
END_IF
bolExecute_old := In_bolExecute;

METHOD FB_exit : BOOL
VAR_INPUT
	bInCopyCode : BOOL; // if TRUE, the exit method is called for exiting an instance that is copied afterwards (online change).
END_VAR
__DELETE(pDelReadPointer);
END_METHOD

METHOD PROTECTED M_AllocMEM : POINTER TO BYTE

VAR_INPUT
	In_SizeOfBuffer : UINT; // Byte size of quee to allocate
END_VAR
// Debug counter
M_AllocMEM := __NEW(BYTE,In_SizeOfBuffer);

// check if allocate memory is ok
IF (M_AllocMEM=TC3_MEMMAN.NULL) THEN
	M_AllocMEM := TC3_MEMMAN.NULL;
ELSE
	Tc2_System.MEMSET(M_AllocMEM,0,In_SizeOfBuffer); // init with zero.
END_IF
END_METHOD

METHOD M_ReleaseAllMEM : BOOL
VAR_INPUT
	In_pstSysInfo : POINTER TO T_FileLc_SysInfo;
END_VAR
VAR
	pDelPointer : POINTER TO BYTE;
END_VAR
// no usage at the moment -> with handle shutdown sequence no easy to remove every thing in the right order


// the other allocated memory has to be deallocated by FB_FileLC! on exit this methode should be called from FB_FileLC!
IF (In_pstSysInfo<>TC3_MEMMAN.NULL) THEN
	__DELETE(In_pstSysInfo^.p_bytHeaderText);
	__DELETE(In_pstSysInfo^.p_bytFooterText);
	FOR ii:=0 TO Queue.cMAX_NR_OF_TASKS BY 1 DO
		IF (In_pstSysInfo^.stItemInfo.a_p_bytItemDataList[ii]<>TC3_MEMMAN.NULL) THEN
			pDelPointer := In_pstSysInfo^.stItemInfo.a_p_bytItemDataList[ii];
			__DELETE(pDelPointer);
			In_pstSysInfo^.stItemInfo.a_p_bytItemDataList[ii] := 0;
		END_IF
	END_FOR
	__DELETE(In_pstSysInfo^.stItemInfo.p_bytItemCfgList);
	__DELETE(In_pstSysInfo^.p_bytTmpRecordText);
	__DELETE(In_pstSysInfo^.stFileHandler.p_bytTmpFileBuffer);
	__DELETE(pDelReadPointer);
END_IF
END_METHOD

END_FUNCTION_BLOCK

// POUs/Utility/strstr
FUNCTION strstr : POINTER TO BYTE
VAR_INPUT
	In_pStr: POINTER TO BYTE; // string which should include search string
	In_pStrSearch: POINTER TO BYTE; // search string
	In_bolAddStrSearchLen : BOOL; // add to result search STRING length
END_VAR
VAR
	p_bytStr : POINTER TO BYTE;
	chrStr : STRING(1) := '';
	p_bytStrSearch : POINTER TO BYTE;
	chrStrSearch : STRING(1) := '';
	ii : UINT;
	jj : UINT;
	p_bytAdressStr : POINTER TO BYTE;
	p_bytAdressStrSearch : POINTER TO BYTE;
END_VAR

(*char *strstr(const char *s1, const char *s2);

Description
Locates the first occurence in the string pointed to by s1 of the sequence of characters in the string pointed to by s2 (excluding the terminating null character). 


Returns
Returns a pointer to the located string segment, or a null pointer if the string s2 is not found. If s2 points to a string with zero length, the s1 is returned. 
*)

// invalid input pointer check
IF ((In_pStr=TC3_MEMMAN.NULL) OR (In_pStrSearch=TC3_MEMMAN.NULL)) THEN
	strstr := TC3_MEMMAN.NULL; // input strings not defined
	RETURN;
END_IF


ii :=0;
p_bytAdressStr := In_pStr;
p_bytStr := p_bytAdressStr;
WHILE (p_bytStr^ <> 0) DO // zero terminated string
	p_bytAdressStr := In_pStr + ii*SIZEOF(In_pStr^); // pointer increment
	p_bytStr := p_bytAdressStr;
	chrStr :=Tc2_System.F_ToCHR(c:= p_bytStr^); // for debugging watch value
	
	jj := 0;
	p_bytAdressStrSearch := In_pStrSearch;
	p_bytStrSearch := p_bytAdressStrSearch;

	WHILE (p_bytStr^ = p_bytStrSearch^) DO
		
		// char/byte matches compare next
		p_bytAdressStrSearch := In_pStrSearch + jj*SIZEOF(In_pStrSearch^); // pointer increment
		p_bytStrSearch := p_bytAdressStrSearch;
		chrStrSearch := Tc2_System.F_ToCHR(c:= p_bytStrSearch^); // for debugging watch value
		
		// end of string found->search string matches
		IF (p_bytStrSearch^=0) THEN// zero terminated string
			IF (In_bolAddStrSearchLen=TRUE) THEN// add to result search STRING length
				strstr := p_bytAdressStr + jj*SIZEOF(In_pStr^); // return start adress of next byte after search string
			ELSE
				strstr := p_bytAdressStr; // return start adress of match search string
			END_IF
			
			RETURN;
		END_IF
		
		p_bytStr := p_bytAdressStr + jj*SIZEOF(In_pStr^);
		chrStr :=Tc2_System.F_ToCHR(c:= p_bytStr^); // for debugging watch value
		jj := jj + 1;
	END_WHILE
	ii := ii + 1;
END_WHILE

strstr := Tc3_MemMan.NULL; // return null adress search string not found in string

END_FUNCTION

// POUs/Utility/Logger/FileLc/FB_FileLcTest
FUNCTION_BLOCK FB_FileLcTest
VAR_INPUT
	In_p_fbBasLog: POINTER TO FB_BasLog; // only one central FB_BasLog instance allowed per PLC!!!
	In_p_fbFileLC: POINTER TO FB_FileLc; // only one central FB_FileLc instance allowed per PLC!!!
	In_strPath: STRING(FileLc.cPATH_LENGTH); //'C:\Vistaprint\Log\'
	In_strCfgFileName: STRING(FileLc.cFILENAME_LENGTH); // 'StateLogTest.cfg'
END_VAR
VAR_OUTPUT
	Out_bolInitDone : BOOL;
	Out_udiStatus : UDINT;
END_VAR
VAR
	bolGetFirstHandle : BOOL;
	bolDone : BOOL;
	udiInitStatus : UDINT;
	udiStatus : UDINT;
	pHandle : POINTER TO T_FileLc_SysInfo;
	// for test send
	pHandleBaseLog : POINTER TO T_Bl_LibHandleRow;
	uinGetHandleBaseLogStatus : UINT;
	intDoWrite : INT;
	dinPar1 : DINT;
	strText1 : STRING(30):='Controller 1';
	strText2 : STRING(30):='Alarm sub info';
	uinWriteStatus : UINT;
	bolStressTest : BOOL;
	fbRAND : DRAND;
	uinActFLcClientIdx : UINT; // file client index for init
END_VAR

(*__________________________________________________________________________________________________
¦	
¦	Vistaprint Schweiz GmbH
¦	CH - 8401 Winterthur
¦
¦	www.vistaprint.ch - info@vistaprint.ch
¦___________________________________________________________________________________________________

Function desription:
Function block capsule the logger file client call for tests.

History:
Version		Date			Author		Comment
---------------------------------------------------------------------------------------------------
0.00.1		27.10.2014		AVME/KVO	Start history
___________________________________________________________________________________________________*)

IF (In_p_fbFileLC<>TC3_MEMMAN.NULL) THEN // check if pointer valid
	
	// system init onetime after start up
	IF (Out_bolInitDone=FALSE) THEN
		In_p_fbFileLC^.M_Init(In_bolExecute := TRUE,In_p_uinFLcIdx := ADR(uinActFLcClientIdx),In_strCfgFileName:=In_strCfgFileName ,In_strPath:= In_strPath,In_p_fbBasLog := In_p_fbBasLog,Out_pHandle=>pHandle,Out_udiStatus=>udiInitStatus,Out_bolDone=>bolDone);
		IF (bolDone OR (udiInitStatus<>0)) THEN
			// negative edge -> reinit possibel and release init next file client!!!
			In_p_fbFileLC^.M_Init(In_bolExecute := FALSE,In_p_uinFLcIdx := ADR(uinActFLcClientIdx),In_strCfgFileName:=In_strCfgFileName,In_strPath:=In_strPath,In_p_fbBasLog := In_p_fbBasLog);
			Out_bolInitDone := TRUE;
		END_IF
	ELSE
		IF ((pHandle<>TC3_MEMMAN.NULL) AND (udiInitStatus=0)) THEN	// valid pointer => init ok
			// cyclic call of file client - alarm generation in application if status not ok???
			udiStatus := In_p_fbFileLC^.M_Cyclic(In_pHandle:=pHandle);
			
			// *******************************************************************************************************************************************
			// only for sending test logs!!!
			// get write handle for tests
			IF (bolGetFirstHandle=FALSE) THEN
				uinGetHandleBaseLogStatus := In_p_fbBasLog^.M_GetHandle(Out_pHandle=>pHandleBaseLog);// fbBasLog global defined base log system fub (only once per system)
				bolGetFirstHandle := TRUE;
			END_IF
			
			// write test state log entries
			IF (pHandleBaseLog<>TC3_MEMMAN.NULL) AND (intDoWrite>0) THEN
				intDoWrite := intDoWrite - 1;
				dinPar1 := dinPar1 + 1;
				uinWriteStatus := In_p_fbBasLog^.M_Log(In_pHandle:=pHandleBaseLog,In_udiLogType:=BasLog.cLOGTYPE_STATELOG,In_intCtrlID:=11,In_strText1:=strText1,In_strText2:=strText2,In_dinPar1:=dinPar1,In_dinPar2:=0,In_dinPar3:=0,In_dinPar4:=0) ;
			END_IF
			IF (bolStressTest) THEN
				IF (intDoWrite = 0) THEN
					fbRAND();
					intDoWrite := LREAL_TO_INT(fbRAND.Num*100.0);
					uinWriteStatus := In_p_fbBasLog^.M_Log(In_pHandle:=pHandleBaseLog,In_udiLogType:=BasLog.cLOGTYPE_STATELOG,In_intCtrlID:=intDoWrite,In_strText1:=strText1,In_strText2:=strText2,In_dinPar1:=dinPar1,In_dinPar2:=0,In_dinPar3:=0,In_dinPar4:=0) ;
				END_IF
			END_IF
			// *******************************************************************************************************************************************
		END_IF;		
	END_IF

	// out for failures
	IF (udiInitStatus<>0)THEN
		Out_udiStatus := udiInitStatus;
	ELSE
		Out_udiStatus := udiStatus;
	END_IF
END_IF

END_FUNCTION_BLOCK

// POUs/Utility/Queue/FB_QueueTest_Receiver
FUNCTION_BLOCK FB_QueueTest_Receiver
VAR_INPUT
	In_p_fbQueue: POINTER TO FB_Queue; // only one central FB_QUEUE instance allowed per PLC!!!
END_VAR
VAR_OUTPUT
END_VAR
VAR
	stData : T_Queue_TestData;
	bolInit : BOOL := FALSE;
	pQueueHandle : POINTER TO T_Queue_SysInfo;
	pQueueHandleRead : POINTER TO T_Queue_Info;
	uinInitStatus : UINT;
	uinGetHandleStatus :UINT;
	uinReadStatus : UINT;
	ii:UINT;
	udiRxCounter : UDINT;
END_VAR

(*__________________________________________________________________________________________________
¦	
¦	Vistaprint Schweiz GmbH
¦	CH - 8401 Winterthur
¦
¦	www.vistaprint.ch - info@vistaprint.ch
¦___________________________________________________________________________________________________

Function desription:
Example and test programm for testing the queue system - read data from queue

History:
Version		Date			Author		Comment
---------------------------------------------------------------------------------------------------
0.00.1		14.07.2014		AVME/KVO	Start history
___________________________________________________________________________________________________*)

// system init onetime after start up
IF (bolInit=FALSE) THEN
	//init queue system, one time should be called per queue system
	In_p_fbQueue^.M_Init(In_strQueueName:='bReceiver',In_uinNrOfElement := 25, In_udiSizeOfElement:= SIZEOF(stData),In_uinMode:=0,Out_pHandle=>pQueueHandle,Out_uinStatus=>uinInitStatus);
	
	// for every task class has to call this methode handle is needed for read
	uinGetHandleStatus := In_p_fbQueue^.M_GetHandle(In_strQueueName:='bReceiver',Out_pQueueHandle=>pQueueHandleRead);
	bolInit := TRUE;
END_IF

// because more than one task function writes to the logsystem it is better to read out more than one elment per cycle!
FOR ii:=0 TO 9 BY 1 DO
	uinReadStatus := In_p_fbQueue^.M_Read(In_pQueueHandle:=pQueueHandleRead,In_pData:=ADR(stData));
	IF (uinReadStatus<>0) THEN
		EXIT;
	END_IF
	udiRxCounter := udiRxCounter + 1;
END_FOR

END_FUNCTION_BLOCK

// POUs/Utility/Queue/FB_QueueTest_Sender
FUNCTION_BLOCK FB_QueueTest_Sender
VAR_INPUT
	In_p_fbQueue: POINTER TO FB_Queue; // only one central FB_QUEUE instance allowed per PLC!!!
END_VAR
VAR_OUTPUT
END_VAR
VAR
	stData : T_Queue_TestData;
	bolInit : BOOL := FALSE;
	pQueueHandle : POINTER TO T_Queue_Info;
	uinGetHandleStatus : UINT;
	uinWriteStatus :UINT;
	uinDoWrite : UINT;
END_VAR

(*__________________________________________________________________________________________________
¦	
¦	Vistaprint Schweiz GmbH
¦	CH - 8401 Winterthur
¦
¦	www.vistaprint.ch - info@vistaprint.ch
¦___________________________________________________________________________________________________

Function desription:
Example and test programm for testing the queue system - write data in queue

History:
Version		Date			Author		Comment
---------------------------------------------------------------------------------------------------
0.00.1		14.07.2014		AVME/KVO	Start history
___________________________________________________________________________________________________*)

// system init onetime after start up
IF (bolInit=FALSE) THEN
	uinGetHandleStatus := In_p_fbQueue^.M_GetHandle(In_strQueueName:='bReceiver',Out_pQueueHandle=>pQueueHandle);
	
	// init write struct
	stData.strName := 'Daten';
	stData.udiAdress := 1;
	stData.udiDataLen := 2;
	stData.usiDataTyp:= 3;
	stData.udiDimension := 4;
	bolInit := TRUE;
END_IF

// number of cycles to write
IF (uinDoWrite>0) THEN
	uinDoWrite := uinDoWrite - 1;
	uinWriteStatus := In_p_fbQueue^.M_Write(In_pQueueHandle:= pQueueHandle,In_pData:= ADR(stData));
	stData.udiAdress := stData.udiAdress + 1;
END_IF

END_FUNCTION_BLOCK

// POUs/Utility/callAllCtrlInit
FUNCTION callAllCtrlInit : BOOL
VAR_INPUT
	pCtrlInst			: POINTER TO POINTER TO FB_CtrlBase;
	uinCtrlInstLength	: UINT;
END_VAR
VAR
	uinIdx	: UINT;
END_VAR

FOR uinIdx := 0 TO uinCtrlInstLength DO
	IF pCtrlInst[uinIdx] <> 0 THEN
		pCtrlInst[uinIdx]^.CtrlInit(); // init ctrl and add childs
	END_IF
END_FOR

END_FUNCTION

// POUs/Utility/getInBol
FUNCTION getInBol : BOOL
VAR_INPUT
	bol_GlobalEnableForce: BOOL;
	p_Input: POINTER TO T_Ctrl_IoBool;
END_VAR

p_Input^.state := p_Input^.map;

IF (p_Input^.EnForce AND bol_GlobalEnableForce) THEN
	p_Input^.intern := p_Input^.force;
ELSE
	p_Input^.intern := p_Input^.map;
END_IF;

getInBol := p_Input^.intern;

END_FUNCTION

// POUs/Utility/getInBolDebounced
FUNCTION getInBolDebounced : BOOL
VAR_INPUT
	bol_GlobalEnableForce: BOOL;
	udiSample_ms: UDINT;		// Sample time from me.FUBInfo.udiSample_ms
	udiDebounceTime_ms: UDINT;	// Wait time for debouncing in ms
	p_Input: POINTER TO T_Ctrl_IoBoolDebounced;
END_VAR

// The input is accepted only after the debounce time (udiDebounceTime_ms)
// If the signal changes during this time, the timer will be restarted

IF (p_Input^.EnForce AND bol_GlobalEnableForce) THEN	// Forced signal, no debouncing neccessary
	p_Input^.intern := p_Input^.force;
ELSE													// Debounce signal
	IF p_Input^.state <> p_Input^.map THEN
		p_Input^.udinDebouncedTimeCounter_ms := 0;
	END_IF
	IF p_Input^.udinDebouncedTimeCounter_ms < udiDebounceTime_ms THEN
		p_Input^.udinDebouncedTimeCounter_ms := p_Input^.udinDebouncedTimeCounter_ms + udiSample_ms;
	ELSE
		p_Input^.intern := p_Input^.map;		
	END_IF
END_IF;

p_Input^.state := p_Input^.map;

getInBolDebounced := p_Input^.intern;

END_FUNCTION

// POUs/Utility/getInInt
FUNCTION getInInt : INT
VAR_INPUT
	bol_GlobalEnableForce: BOOL;
	p_Input: POINTER TO T_Ctrl_IoInt;
END_VAR

p_Input^.state := p_Input^.map;

IF (p_Input^.EnForce AND bol_GlobalEnableForce) THEN
	p_Input^.intern := p_Input^.force;
ELSE
	p_Input^.intern := p_Input^.map;
END_IF;

getInInt := p_Input^.intern;

END_FUNCTION

// POUs/Utility/getInUint
FUNCTION getInUint : UINT
VAR_INPUT
	bol_GlobalEnableForce		: BOOL;
	p_Input						: POINTER TO T_Ctrl_IoUint;
END_VAR
VAR
END_VAR

p_Input^.state := p_Input^.map;

IF (p_Input^.EnForce AND bol_GlobalEnableForce) THEN
	p_Input^.intern := p_Input^.force;
ELSE
	p_Input^.intern := p_Input^.map;
END_IF;

getInUint := p_Input^.intern;

END_FUNCTION

// POUs/Utility/getInUsint
FUNCTION getInUsint : USINT
VAR_INPUT
	bol_GlobalEnableForce		: BOOL;
	p_Input						: POINTER TO T_Ctrl_IoUsint;
END_VAR
VAR
END_VAR

p_Input^.state := p_Input^.map;

IF (p_Input^.EnForce AND bol_GlobalEnableForce) THEN
	p_Input^.intern := p_Input^.force;
ELSE
	p_Input^.intern := p_Input^.map;
END_IF;

getInUsint := p_Input^.intern;

END_FUNCTION

// POUs/Utility/initAllCtrl
FUNCTION initAllCtrl : BOOL
VAR_INPUT
	pCtrlInst			: POINTER TO POINTER TO FB_CtrlBase;
	pBasLogFB			: POINTER TO FB_BasLog;
	pAlarmCtrl			: POINTER TO FB_Alm_Man;
	uinCtrlInstLength	: UINT;
END_VAR
VAR
	uinIdx	: UINT;
END_VAR

FOR uinIdx := 0 TO uinCtrlInstLength DO
	IF pCtrlInst[uinIdx] <> 0 THEN
		IF (pAlarmCtrl<>0) THEN
			pCtrlInst[uinIdx]^.AlarmCtrl := pAlarmCtrl; // add alarm manager interface/pointer
		END_IF
		IF (pBasLogFB<>0) THEN
			pCtrlInst[uinIdx]^.BaseLog := pBasLogFB; // add base logger interface/pointer
		END_IF
		pCtrlInst[uinIdx]^.CtrlInit(); // init ctrl and add childs
	END_IF
END_FOR

END_FUNCTION

// POUs/Utility/ScaleINT
FUNCTION ScaleINT : INT //Output signal.
VAR_INPUT
	x: INT; 	// Input signal. Allowed values: -32768..+32767.
	x1 : INT;	// Abscissa for the 1st coordinate. Allowed values: -32768..+32767
	x2 : INT;	// Abscissa for the 2nd coordinate. Allowed values: -32768..+32767.
	y1 : INT;	// Ordinate for the 1st coordinate. First limit of the value range. Allowed values: –32768..+32767.
	y2: INT;	// Ordinate for the 2nd coordinate. Second limit of the value range. Allowed values: -32768..+32767.
END_VAR
VAR
END_VAR


(*	IF x1 = x2, THEN 0 is output *)

// Scale value 
IF (x1=x2) THEN // -> zero division!
	ScaleINT := 0;
ELSE
	ScaleINT := (((x - x1) * (y2-y1))/(x2-x1)) + y1;
END_IF

END_FUNCTION

// POUs/Utility/setAllCtrlAlarmFB
FUNCTION setAllCtrlAlarmFB : BOOL
VAR_INPUT
	pCtrlInst			: POINTER TO POINTER TO FB_CtrlBase;
	pAlarmCtrl			: POINTER TO FB_Alm_Man;
	uinCtrlInstLength	: UINT;
END_VAR
VAR
	uinIdx	: UINT;
END_VAR

FOR uinIdx := 0 TO uinCtrlInstLength DO
	IF pCtrlInst[uinIdx] <> 0 THEN
		pCtrlInst[uinIdx]^.AlarmCtrl := pAlarmCtrl;
	END_IF
END_FOR

END_FUNCTION

// POUs/Utility/setAllCtrlBasLogFB
FUNCTION setAllCtrlBasLogFB : BOOL
VAR_INPUT
	pCtrlInst			: POINTER TO POINTER TO FB_CtrlBase;
	pBasLogFB			: POINTER TO FB_BasLog;
	uinCtrlInstLength	: UINT;
END_VAR
VAR
	uinIdx	: UINT;
END_VAR

FOR uinIdx := 0 TO uinCtrlInstLength DO
	IF pCtrlInst[uinIdx] <> 0 THEN
		pCtrlInst[uinIdx]^.BaseLog := pBasLogFB;
	END_IF
END_FOR

END_FUNCTION

// POUs/Utility/setOutBol
FUNCTION setOutBol : BOOL
VAR_INPUT
	bol_GlobalEnableForce: BOOL;
	p_Output: POINTER TO T_Ctrl_IoBool;
END_VAR

// Copy real values
p_Output^.state := p_Output^.intern;

IF (p_Output^.EnForce AND bol_GlobalEnableForce) THEN
	p_Output^.map := p_Output^.force;
ELSE
	p_Output^.map := p_Output^.intern;
END_IF;

setOutBol := p_Output^.map;

END_FUNCTION

// POUs/Utility/setOutInt
FUNCTION setOutInt : INT
VAR_INPUT
	bol_GlobalEnableForce: BOOL;
	p_Output: POINTER TO T_Ctrl_IoInt;
END_VAR

// Copy real values
p_Output^.state := p_Output^.intern;

IF (p_Output^.EnForce AND bol_GlobalEnableForce) THEN
	p_Output^.map := p_Output^.force;
ELSE
	p_Output^.map := p_Output^.intern;
END_IF;

setOutInt := p_Output^.map;

END_FUNCTION

// POUs/Utility/setOutUint
FUNCTION setOutUint : UINT
VAR_INPUT
	bol_GlobalEnableForce	: BOOL;
	p_Output				: POINTER TO T_Ctrl_IoUint;
END_VAR
VAR
END_VAR

// Copy real values
p_Output^.state := p_Output^.intern;

IF (p_Output^.EnForce AND bol_GlobalEnableForce) THEN
	p_Output^.map := p_Output^.force;
ELSE
	p_Output^.map := p_Output^.intern;
END_IF;

setOutUint := p_Output^.map;

END_FUNCTION

// POUs/Utility/setOutUsint
FUNCTION setOutUsint : USINT
VAR_INPUT
	bol_GlobalEnableForce	: BOOL;
	p_Output				: POINTER TO T_Ctrl_IoUsint;
END_VAR
VAR
END_VAR

// Copy real values
p_Output^.state := p_Output^.intern;

IF (p_Output^.EnForce AND bol_GlobalEnableForce) THEN
	p_Output^.map := p_Output^.force;
ELSE
	p_Output^.map := p_Output^.intern;
END_IF;

setOutUsint := p_Output^.map;

END_FUNCTION
